Omron Sysmac Studio project TlsClientLib (Sysmac Studio 1.62.0.9, LibraryProject)
(* Develop simple TLS client library. *)

# Controller LIB: NX102-9000 version 1.64
Task Subsystem (priority 18, period or condition 10000): Example_SendLog
Library RingBufferLib 0.0.2 (contents left out)

TYPE stfreakjp\net\TlsClientContext : STRUCT
    Busy : BOOL;
    Active : BOOL;
    Error : BOOL;
    ErrorID : WORD;
    ErrorIDEx : DWORD;
    Port : UINT;
    Destination : STRING[256];
    DestinationPort : UINT;
    TLSSessionName : STRING[16];
    UseRecv : BOOL;
    UseSend : BOOL;
    UseWatcher : BOOL;
    UseTcpSocketOption : BOOL;
    OptionNodelay : BOOL;
    ConnectRetryTimes : UINT;
    ConnectRetryInterval : UINT;
    ConnectTimeout : UINT;
    WatchInterval : UINT;
    CtrlActive : BOOL;
    CtrlAllowSend : BOOL;
    CtrlAllowRecv : BOOL;
    Socket : _sSOCKET;
    TLSHandle : DWORD;
    Reconnecting : BOOL;
    Connected : BOOL;
    SendTimes : ULINT;
    SendSize : ULINT;
    RecvTimes : ULINT;
    RecvSize : ULINT;
END_STRUCT END_TYPE

PROGRAM README
RETURN;
(*

# About This Project
This project is for the development of the stream-oriented TLS clients: TlsClient, TlsSendClient, and TlsRecvClient.
TlsClient reads and writes TLS send/receive data to and from a ring buffer passed as a parameter.

The ring buffer utilizes RingBufferLib.
RingBufferLib is an implementation of a ring buffer for BYTE type arrays.
The RingBufferLib implementation can be used in multi-tasking environments without needing locks,
but only when there is a single reader and a single writer to the buffer.
TlsClient inherits this characteristic.

# About the Programs
This project includes the following examples.

* POU/Program/Example_SendLog
  This program uses TlsClient to send the contents of a logger's buffer to a remote location.
  Additionally, a debug-purpose TlsClient runs,
  monitoring and remotely sending the transmit buffer of the TlsClient that sends the logs.

Please refer to each program for usage steps.


# このプロジェクトについて
このプロジェクトは、ストリーム型TLSクライアントであるTlsClient/TlsSendClient/TlsRecvClientの開発用プロジェクトです。
TlsClientは、パラメータとして渡したリングバッファに対してTLSによる送受信データを読み書きします。
リングバッファは、RingBufferLibを使用します。
RingBufferLibはBYTE型配列を対象とするリングバッファの実装です。
RingBufferLibの実装は、バッファへの読み書きの主体がそれぞれ1つである時に限り、ロックを使用しなくてもマルチタスクに使用することができます。
TlsClientはその特性を引き継ぎます。

# プログラムについて
このプロジェクトは、以下の使用例を含みます。

* POU/プログラム/Example_SendLog
  TlsClientを使用してロガーのバッファ内容をリモートに送信します。
  また、ログを送信するTlsClientの送信バッファを監視してリモートに送信するデバッグ用のTlsClientが動作します。

使用手順については、各プログラムを確認してください。


For the parts to which I have rights, I follow POU/Program/LICENSE.
You are free to use and modify it, but we are not responsible for any damage or loss related to it.

(c) 2025 KITA Munemitsu

*)
END_PROGRAM

PROGRAM Example_SendLog
VAR CONSTANT
    LOG_SENDER_RESET_PAYLOAD : STRING[8] := '$$R$$L$$R$$L';
END_VAR
VAR
    REMOTE_ADDR : STRING[256];
    REMOTE_PORT : UINT;
    SPY_REMOTE_PORT : UINT;
    DEBUG_WRITE_REMOTE_PORT : UINT;
    DEBUG_READ_REMOTE_PORT : UINT;
    LOGGING_INTERVAL : UINT;
    iLogSenderTlsClient : stfreakjp\net\TlsClient;
    iLogSenderContext : stfreakjp\net\TlsClientContext;
    iLogSenderSendBufferContext : stfreakjp\buf\RingBufferContext;
    iLogSenderSendBuffer : ARRAY[0..8191] OF BYTE;
    iLogSenderRecvBufferContext : stfreakjp\buf\RingBufferContext;
    iLogSenderRecvBuffer : ARRAY[0..8191] OF BYTE;
    iLoggerWrittenTracker : stfreakjp\buf\RingBufferContext;
    iLoggerBufferContext : stfreakjp\buf\RingBufferContext;
    iLoggerBuffer : ARRAY[0..4095] OF BYTE;
    iPayload : ARRAY[0..4095] OF BYTE;
    iPayloadSize : UINT;
    iMsg : STRING[1024];
    iWaitTick : UINT;
    iSpySenderTlsClient : stfreakjp\net\TlsSendClient;
    iSpySenderClientContext : stfreakjp\net\TlsClientContext;
    iSpySendBufferContext : stfreakjp\buf\RingBufferContext;
    iSpySendBuffer : ARRAY[0..8191] OF BYTE;
    iSpyLogSenderSentTracker : stfreakjp\buf\RingBufferContext;
    iDebugReadSenderTlsClient : stfreakjp\net\TlsSendClient;
    iDebugReadSenderClientContext : stfreakjp\net\TlsClientContext;
    iDebugWriteSenderTlsClient : stfreakjp\net\TlsSendClient;
    iDebugWriteSenderClientContext : stfreakjp\net\TlsClientContext;
    iDebugWriteSenderBufferContext : stfreakjp\buf\RingBufferContext;
    iDebugWriteSenderBuffer : ARRAY[0..19999] OF BYTE;
    iDebugReadSenderBufferContext : stfreakjp\buf\RingBufferContext;
    iDebugReadSenderBuffer : ARRAY[0..19999] OF BYTE;
    iDebugLogSenderSendTracker : stfreakjp\buf\RingBufferContext;
    iToggleLogSend : BOOL;
END_VAR
(*

# About This Program
This program uses TlsClient to send the contents of a logger's buffer to a remote location.
Additionally, a debug-purpose TlsClient runs,
monitoring and remotely sending the transmit buffer of the TlsClient that sends the logs.

It is composed of the following:

* A logger that continuously writes logs.
* A log sender that sends logs written by the logger via TLS.
* A spy sender that monitors the log sender's transmission buffer and sends potentially transmitted logs via TLS.
* A debug sender that monitors read/write operations of the log sender's transmission buffer and sends each change via TLS.

# Usage Steps
Follow these steps to use the program.

1.  Adjust the project configuration to match your operating environment.   
    Match the controller model and ensure access to the network you intend to use.
  
2.  Adjust `POU/Program/Example_SendLog` to match your operating environment.   
    Change the value of the `REMOTE_ADDR` variable to the address of the device waiting for data.

3.  Start TLS endpoints on an appropriate device and wait for connections.
    You can find a reference PowerShell script in `POU/Program/SimpleTlsMonitor_ps1`.
	`StartMultiMonitors_ps1` is a PowerShell script that uses Windows Terminal to launch four TLS endpoints.

4.  Register TLS sessions on the controller.
    Register four TLS sessions with IDs 0-3.

5.  Run the program on the controller.   
    Transfer the program to the controller and start its execution.

6.  Confirm that data is sent to the listening TLS endpoints.


# このプログラムについて
このプログラムは、TlsClientを使用してロガーのバッファ内容をリモートに送信します。
また、ログを送信するTlsClientの送信バッファを監視してリモートに送信するデバッグ用のTlsClientが動作します。

以下によって構成します。

* ログを書き込み続けるロガー
* ロガーが書き込んだログをTLSで送信するログ送信クライアント
* ログ送信クライアントの送信バッファを監視して送信した可能性のあるログをTLSで送信するスパイ送信クライアント
* ログ送信クライアントの送信バッファの読み書きを監視して、それぞれの変化をTLSで送信するデバッグ送信クライアント

# 使用手順
このプログラムは、以下の手順で使用します。

1.  プロジェクトの構成を使用環境に合わせる
    コントローラの型式を合わせ、使用するネットワークにアクセスできるようにします。
  
2.  `POU/プログラム/Example_SendLog`を使用環境に合わせる
    `REMOTE_ADDR`変数の値をデータを待ち受ける端末のアドレスに変更します。
  
3.  適当な端末にTLSエンドポイントを立ち上げ待ち受ける
    `POU/プログラム/SimpleTlsMonitor_ps1`に参考のPowerShellスクリプトがあります。
	`StartMultiMonitors_ps1`は、Windows Terminalを使用して4つのTLSエンドポイントを立ち上げるPowerShellスクリプトです。

4.  コントローラにTLSセッションを登録する
    4つのTLSセッションをID 0-3で登録します。

5.  コントローラでプログラムを動作させる
    プログラムをコントローラに転送して動作させます。
  
6.  待ち受けているTLSエンドポイントにデータが送られてくることを確認する


(c) 2025 KITA Munemitsu

*)

// Change according to your environment.
IF P_First_Run THEN
	REMOTE_ADDR := 'YOUR_REMOTE_DEVICE';
	REMOTE_PORT := 12101;
	SPY_REMOTE_PORT := 12102;
	DEBUG_WRITE_REMOTE_PORT := 13101;
	DEBUG_READ_REMOTE_PORT := 13102;
	LOGGING_INTERVAL := 1;
END_IF;

IF P_First_Run THEN	
	// Setup Logger.
	Logger_init(Context:=iLoggerBufferContext,
				Buffer:=iLoggerBuffer);	

	// Setup Log sender.
	//
	// The log sender monitors the logger buffer and sends the written logs.
	//
	RingBuffer_init(Context:=iLogSenderSendBufferContext,
					Buffer:=iLogSenderSendBuffer);
	RingBuffer_init(Context:=iLogSenderRecvBufferContext,
					Buffer:=iLogSenderRecvBuffer);
	TlsClient_configure(Context:=iLogSenderContext,
						Activate:=TRUE,
						Destination:=REMOTE_ADDR,
						DestinationPort:=REMOTE_PORT,
						Port:=0,
						TLSSessionName:='TLSSession0',
						UseSend:=TRUE,
						UseRecv:=FALSE,
						UseWatcher:=TRUE,
						WatchInterval:=600,
						ConnectRetryTimes:=100,
						ConnectRetryInterval:=600);
	iLogSenderTlsClient.Enable := TRUE;
	// Tracks logger writes.
	RingBuffer_createWriteTracker(Target:=iLoggerBufferContext,
								  Tracker=>iLoggerWrittenTracker);

	// Setup Spy sender.
	//
    // The spy monitors the sender's transmit buffer and transmits any data that may have been sent.
	//
	RingBuffer_init(Context:=iSpySendBufferContext,
					Buffer:=iSpySendBuffer);
	TlsClient_configure(Context:=iSpySenderClientContext,
						Activate:=TRUE,
						Destination:=REMOTE_ADDR,
						DestinationPort:=SPY_REMOTE_PORT,
						Port:=0,
						TLSSessionName:='TLSSession1',
						UseSend:=TRUE,
						UseWatcher:=TRUE,
						WatchInterval:=600,
						ConnectRetryTimes:=100,
						ConnectRetryInterval:=600);
	iSpySenderTlsClient.Enable := TRUE;
	// Tracks reads of the log sender's send buffer.
	RingBuffer_createReadTracker(Target:=iLogSenderSendBufferContext,
								 Tracker=>iSpyLogSenderSentTracker);
 
    // Setup Debug senders.
	//
	// The debug sender monitors the input and output of the log sender's send buffer and sends the changes.
	//
	RingBuffer_init(Context:=iDebugWriteSenderBufferContext,
					Buffer:=iDebugWriteSenderBuffer);
	TlsClient_configure(Context:=iDebugWriteSenderClientContext,
						Activate:=TRUE,
						Destination:=REMOTE_ADDR,
						DestinationPort:=DEBUG_WRITE_REMOTE_PORT,
						Port:=0,
						TLSSessionName:='TLSSession2',
						UseSend:=TRUE,
						WatchInterval:=600,
						ConnectRetryTimes:=100,
						ConnectRetryInterval:=600);
	iDebugWriteSenderTlsClient.Enable := TRUE;
	
	RingBuffer_init(Context:=iDebugReadSenderBufferContext,
					Buffer:=iDebugReadSenderBuffer);
	TlsClient_configure(Context:=iDebugReadSenderClientContext,
						Activate:=TRUE,
						Destination:=REMOTE_ADDR,
						DestinationPort:=DEBUG_READ_REMOTE_PORT,
						Port:=0,
						TLSSessionName:='TLSSession3',
						UseSend:=TRUE,
						WatchInterval:=600,
						ConnectRetryTimes:=100,
						ConnectRetryInterval:=600);
	iDebugReadSenderTlsClient.Enable := TRUE;
	// Tracks the log sender's send buffer in and out.
	RingBuffer_createTracker(Target:=iLogSenderSendBufferContext,
							 Tracker=>iDebugLogSenderSendTracker);

	// Sends the log sender reset payload first.
	RingBuffer_writeString(Context:=iLogSenderSendBufferContext,
						   Buffer:=iLogSenderSendBuffer,
						   Value:=LOG_SENDER_RESET_PAYLOAD);

	iWaitTick := LOGGING_INTERVAL;
END_IF;

// Logging at regular intervals.
Dec(iWaitTick);
IF iWaitTick < 1 THEN
	iMsg := CONCAT('{"counter":', ULINT_TO_STRING(Get1usCnt()),
				   ',"timestamp":"', DtToString(GetTime()),
				   '"}$L');
	Logger_write(Context:=iLoggerBufferContext,
				 Buffer:=iLoggerBuffer,
				 Message:=iMsg);
	
	iWaitTick := LOGGING_INTERVAL;
END_IF;

IF iToggleLogSend THEN
	IF TlsClient_isAllowSend(Context:=iLogSenderContext) THEN
		TlsClient_disallowSend(Context:=iLogSenderContext);
	ELSE
		TlsClient_allowSend(Context:=iLogSenderContext);
	END_IF;
	iToggleLogSend := FALSE;
END_IF;

// Gets the difference of the logger buffer into the log sender's send buffer.
RingBuffer_pullWrite(Context:=iLogSenderSendBufferContext,
					 Buffer:=iLogSenderSendBuffer,
					 Tracker:=iLoggerWrittenTracker,
					 Tracked:=iLoggerBufferContext,
					 TrackedBuffer:=iLoggerBuffer);
iLogSenderTlsClient(Context:=iLogSenderContext,
					SendBufferContext:=iLogSenderSendBufferContext,
					SendBuffer:=iLogSenderSendBuffer,
					RecvBufferContext:=iLogSenderRecvBufferContext,
					RecvBuffer:=iLogSenderRecvBuffer);

// Gets the difference between the read data in the log sender's send buffer.
RingBuffer_pullRead(Context:=iSpySendBufferContext,
					Buffer:=iSpySendBuffer,
					Tracker:=iSpyLogSenderSentTracker,
					Tracked:=iLogSenderSendBufferContext,
					TrackedBuffer:=iLogSenderSendBuffer);
iSpySenderTlsClient(Context:=iSpySenderClientContext,
					SendBufferContext:=iSpySendBufferContext,
					SendBuffer:=iSpySendBuffer);

// Gets the read and write deferences of the log sender's send buffer.
RingBuffer_pull(WriteContext:=iDebugWriteSenderBufferContext,
				WriteBuffer:=iDebugWriteSenderBuffer,
				ReadContext:=iDebugReadSenderBufferContext,
				ReadBuffer:=iDebugReadSenderBuffer,
				Tracker:=iDebugLogSenderSendTracker,
				Tracked:=iLogSenderSendBufferContext,
				TrackedBuffer:=iLogSenderSendBuffer);
iDebugWriteSenderTlsClient(Context:=iDebugWriteSenderClientContext,
						   SendBufferContext:=iDebugWriteSenderBufferContext,
						   SendBuffer:=iDebugWriteSenderBuffer);
iDebugReadSenderTlsClient(Context:=iDebugReadSenderClientContext,
						  SendBufferContext:=iDebugReadSenderBufferContext,
						  SendBuffer:=iDebugReadSenderBuffer);
END_PROGRAM

PROGRAM SimpleTlsMonitor_ps1
RETURN;
(*

Below is a PowerShell script that starts a TLS server and waits for clients.


以下は、TLSサーバを立ち上げてクライアントを待ち受けるPowerShellスクリプトです。

```powershell:simple-tls-monitor.ps1
param(
    [Parameter(Mandatory=$false, Position=0)][int]$Port = 12101,
    [Parameter(Mandatory=$false, Position=1)][int]$ReadInterval = 50,
    [Parameter(Mandatory=$false, Position=2)][string]$Mode = 'jsonl',
    [Parameter(Mandatory=$false, Position=3)][string]$CertFriendlyName = 'TlsClientLibTest'
)

# Modify the following script and run it in PowerShell with administrator privileges
# to create a self-signed certificate.
#
# $param = @{
#    Type = 'SSLServerAuthentication'
#    DnsName = 'SET_YOUR_DOMAIN'
#    CertStoreLocation = 'Cert:\CurrentUser\My'
#    FriendlyName = 'TlsClientLibTest'
# }
# New-SelfSignedCertificate @params
#

$serverCert = Get-ChildItem -Path Cert:\CurrentUser\My
        | Where-Object { $_.FriendlyName -eq $CertFriendlyName }
if ($null -eq $serverCert) {
    Write-Host "No certs."
}

function Mode-Jsonl {
    param(
        [int]$Port,
        [int]$ReadInterval,
        [Object]$cert
    )
    $listenerEndPoint = New-Object IPEndpoint([System.Net.IPAddress]::Any, $Port)
    $tcpListener = New-Object System.Net.Sockets.TCPListener($listenerEndpoint)
    $client = $null
    $clientStream = $null
    $sslStream = $null
    $reader = $null
    $task = $null
    $entity = $null
    $prevEntity = $null

    try {
        $tcpListener.Start()
        while ($true) {
            # Wait for client connection.
            if ($null -eq $client) {
                if ($null -eq $task) {
                    $task = $tcpListener.AccepttcpClientAsync()
                }
                if (-not $task.Wait(200)) {
                    continue
                }
                $client = $task.GetAwaiter().GetResult()
                $clientStream = $client.GetStream()
                $sslStream = New-Object System.Net.Security.SslStream($clientStream, $false)
                $sslStream.AuthenticateAsServerAsync($cert, $false, [System.Security.Authentication.SslProtocols]::Tls12, $false).Wait()

                $reader = New-Object System.IO.StreamReader($sslStream)
                $task = $null
            }
            if ($reader.EndOfStream) {
                $reader.Close()
                $sslStream.Close()
                $clientStream.Close()
                $client.Close()
                $task = $null
                $reader = $null
                $clientStream = $null
                $client = $null
                $entity = $null
                $prevEntity = $null
                continue
            }

            # Waiting to receive data.
            try {
                if ($null -eq $task) {
                    $task = $reader.ReadLineAsync()
                }

                if (-not $task.Wait($ReadInterval)) {
                    continue
                }
                $entity = $task.GetAwaiter().GetResult();
                $task = $null
            }
            catch {
                Write-Host "error: $($_.Exception.Message)"
                $reader.Close()
                $clientStream.Close()
                $client.Close()
                $reader = $null
                $ClientStream = $null
                $client = $null
            }

            if ($null -ne $entity) {
                if ("" -eq $entity) {
                    if ("" -eq $prevEntity) {
                        Write-Host 'reset'
                    }
                } else {
                    try {
                        $entity | ConvertFrom-Json | Write-Host
                    }
                    catch {
                        Write-Host "error payload: ${entity}"
                    }
                }
            }

            $prevEntity = $entity
            $entity = $null
        }
    }
    catch {
        Write-Host "error: $($_.Exception.Message)"
    }
    finally {
        if ($client) {
            $reader.Close()
            $sslStream.Close()
            $clientStream.Close()
            $client.Close()
        }
        $tcpListener.Stop()
    }
}

function Mode-Raw {
    param(
        [string]$Port,
        [int]$ReadInterval,
        [Object]$cert
    )
    $listenerEndPoint = New-Object IPEndpoint([System.Net.IPAddress]::Any, $Port)
    $tcpListener = New-Object System.Net.Sockets.TCPListener($listenerEndpoint)
    $client = $null
    $clientStream = $null
    $reader = $null
    $task = $null
    $prevEntity = $null

    try {
        $tcpListener.Start()
        while ($true) {
            # Wait for client connection.
            if ($null -eq $client) {
                if ($null -eq $task) {
                    $task = $tcpListener.AcceptTcpClientAsync()
                }
                if (-not $task.Wait(200)) {
                    continue
                }

                $client = $task.GetAwaiter().GetResult();
                $clientStream = $client.GetStream()
                $sslStream = New-Object System.Net.Security.SslStream($clientStream, $false)
                $sslStream.AuthenticateAsServer($cert, $false, [System.Security.Authentication.SslProtocols]::Tls12, $false)
                $reader = New-Object System.IO.StreamReader($sslStream)
                $task = $null
            }
            if ($reader.EndOfStream) {
                $reader.Close()
                $sslStream.Close()
                $clientStream.Close()
                $client.Close()
                $task = $null
                $reader = $null
                $clientStream = $null
                $client = $null
                $entity = $null
                $prevEntity = $null
                continue
            }

            # Waiting to receive data.
            try {
                if ($null -eq $task) {
                    $task = $reader.ReadLineAsync()
                }

                if (-not $task.Wait($ReadInterval)) {
                    continue
                }
                $entity = $task.GetAwaiter().GetResult();
                $task = $null
            }
            catch {
                Write-Host "error: $($_.Exception.Message)"
                $reader.Close()
                $sslStream.Close()
                $clientStream.Close()
                $client.Close()
                $reader = $null
                $sslStream = $null
                $ClientStream = $null
                $client = $null
            }

            if ($null -ne $entity) {
                if ("" -eq $entity) {
                    if ("" -eq $prevEntity) {
                        Write-Host 'reset'
                    }
                } else {
                    $entity | Write-Host
                }
            }

            $prevEntity = $entity
            $entity = $null
        }
    }
    catch {
        Write-Host "error: $($_.Exception.Message)"
    }
    finally {
        if ($client) {
            $reader.Close()
            $sslStream.Close()
            $clientStream.Close()
            $client.Close()
        }
        $tcpListener.Stop()
    }
}

switch ( $Mode )
{
    Jsonl { Mode-Jsonl -Port $Port -ReadInterval $ReadInterval -cert $serverCert }
    Raw   { Mode-Raw -Port $Port -ReadInterval $ReadInterval -cert $serverCert }
}
```
*)
END_PROGRAM

PROGRAM StartMultiMonitors_ps1
RETURN;
(*

Below is a PowerShell script that launches four "simple-tls-monitor.ps" files in Windows Terminal.
Run this script while "simple-tls-monitor.ps1" is in the same folder.


以下は、Windows Terminalで4つの"simple-tls-monitor.ps"を立ち上げるPowerShellスクリプトです。
"simple-tls-monitor.ps1"が同じフォルダにある状態で実行します。

```powershell:start-multi-monitors.ps1
param(
    [Parameter(Mandatory=$false, Position=0)][int[]]$Ports = @(12101, 12102, 13101, 13102),
    [Parameter(Mandatory=$false, Position=1)][string]$Mode = 'jsonl',
    [Parameter(Mandatory=$false, Position=3)][string]$CertFriendlyName = 'TlsClientLibTest'
)

$scriptFile = "simple-tls-monitor.ps1"
$scriptDir = Split-Path -Parent $MyInvocation.MyCommand.Definition
$scriptPath = Join-Path $scriptDir $scriptFile
if (-not (Test-Path $scriptPath)) {
    Write-Error "error: Not fount '${scriptFile}' in '${scriptPath}'"
    exit 1
}

$wtCommandString = "pwsh.exe -NoExit -Command ""&{ & `"${scriptPath}`" -Port $($Ports[0]) -Mode `"${Mode}`" -CertFriendlyName `"${CertFriendlyName}`" }"" ; " + `
                   "split-pane -H pwsh.exe -NoExit -Command ""&{ & `"${scriptPath}`" -Port $($Ports[1]) -Mode `"${Mode}`" -CertFriendlyName `"${CertFriendlyName}`" }"" ; " + `
                   "split-pane -V pwsh.exe -NoExit -Command ""&{ & `"${scriptPath}`" -Port $($Ports[2]) -Mode `"${Mode}`" -CertFriendlyName `"${CertFriendlyName}`" }"" ; " + `
                   "split-pane -H pwsh.exe -NoExit -Command ""&{ & `"${scriptPath}`" -Port $($Ports[3]) -Mode `"${Mode}`" -CertFriendlyName `"${CertFriendlyName}`" }"""

# For debug.
# Write-Host "command: wt.exe $wtCommandString"

Start-Process -FilePath "wt.exe" -ArgumentList $wtCommandString
```
*)
END_PROGRAM

PROGRAM LICENSE
RETURN;
(*
The MIT License (MIT)

Copyright(c) 2025 KITA Munemitsu

Permission is hereby granted, free of charge, to any person obtaining a copy of this software and associated
documentation files (the “Software”), to deal in the Software without restriction, including without limitation
the rights to use, copy, modify, merge, publish, distribute, sublicense, and/or sell copies of the Software,
and to permit persons to whom the Software is furnished to do so, subject to the following conditions:

The above copyright notice and this permission notice shall be included in all copies or substantial portions of the Software.

THE SOFTWARE IS PROVIDED “AS IS”, WITHOUT WARRANTY OF ANY KIND, EXPRESS OR IMPLIED, INCLUDING BUT NOT
LIMITED TO THE WARRANTIES OF MERCHANTABILITY, FITNESS FOR A PARTICULAR PURPOSE AND NONINFRINGEMENT.
IN NO EVENT SHALL THE AUTHORS OR COPYRIGHT HOLDERS BE LIABLE FOR ANY CLAIM, DAMAGES OR OTHER LIABILITY,
WHETHER IN AN ACTION OF CONTRACT, TORT OR OTHERWISE, ARISING FROM, OUT OF OR IN CONNECTION WITH THE SOFTWARE
OR THE USE OR OTHER DEALINGS IN THE SOFTWARE.
*)
END_PROGRAM

FUNCTION stfreakjp\net\TlsClient_configure : BOOL
(* Initializes the TlsClientContext. *)
VAR_IN_OUT
    Context : stfreakjp\net\TlsClientContext;
END_VAR
VAR_INPUT
    Activate : BOOL := True;  (* Whether to activate the TLS client. Default is TRUE. *)
    Destination : STRING[256] := '';  (* Destination address. *)
    DestinationPort : UINT := 12101;  (* Destination port number. Default is 12101. *)
    Port : UINT := 0;  (* Port number of the TLS client socket. Default is 0 (Auto). *)
    TLSSessionName : STRING[16] := 'TLSSession0';  (* TLSSession name. Default is "TLSSession0". *)
    UseSend : BOOL := False;  (* Whether to use the Send feature. Default is FALSE. *)
    UseRecv : BOOL := False;  (* Whether to use the receive feature. Default is FALSE. *)
    UseWatcher : BOOL := False;  (* Whether to periodically check the connection status. Default is FALSE. *)
    WatchInterval : UINT := 300;  (* Interval between connection status checks. In 100ms increments. Defalt is 300 (30 sec). *)
    ConnectRetryTimes : UINT := 100;  (* Number of times the reconnect process will be attempted. Default is 100. *)
    ConnectRetryInterval : UINT := 300;  (* Interval between reconnection attempts. In 100ms increments. Defalt is 100 (10 sec). *)
    ConnectTimeout : UINT := 50;  (* Timeout waiting for connection. In 100ms increments. Default is 50 (5 sec). *)
    OptionNodelay : BOOL := False;  (* TCP_NODELAY option value. Default is FALSE. *)
END_VAR
(*

Initializes the TlsClientContext.


TlsClientContextを初期化する。


(c) 2025 KITA Munemitsu

*)

IF NOT EN THEN
	TlsClient_configure := FALSE;
	
	RETURN;
END_IF;

Context.CtrlActive := Activate;
Context.CtrlAllowSend := UseSend;
Context.CtrlAllowRecv := UseRecv;
Context.Destination := Destination;
Context.DestinationPort := DestinationPort;
Context.Port := Port;
Context.TLSSessionName := TLSSessionName;
Context.UseSend := UseSend;
Context.UseRecv := UseRecv;
Context.UseWatcher := UseWatcher;
Context.ConnectRetryTimes := ConnectRetryTimes;
Context.ConnectRetryInterval := ConnectRetryInterval;
Context.ConnectTimeout := ConnectTimeout;
Context.WatchInterval := WatchInterval;
Context.UseTcpSocketOption := OptionNodelay;
Context.OptionNodelay := OptionNodelay;

TlsClient_configure := TRUE;
END_FUNCTION

FUNCTION stfreakjp\net\TlsClient_activate : BOOL
(* Activates the TLS client. *)
VAR_IN_OUT
    Context : stfreakjp\net\TlsClientContext;  (* Target TlsClientContext. *)
END_VAR
(*

Activates the TLS client.


TLSクライアントを有効化する。


(c) 2025 KITA Munemitsu

*)

IF NOT EN THEN
	TlsClient_activate := FALSE;
	
	RETURN;
END_IF;
TlsClient_activate := TRUE;

Context.CtrlActive := TRUE;
END_FUNCTION

FUNCTION stfreakjp\net\TlsClient_deactivate : BOOL
(* Deactivates the TLS client. *)
VAR_IN_OUT
    Context : stfreakjp\net\TlsClientContext;  (* Target TlsClientContext. *)
END_VAR
(*

Deactivates the TLS client.


TLSクライアントを無効化する。


(c) 2025 KITA Munemitsu

*)

IF NOT EN THEN
	TlsClient_deactivate := FALSE;
	
	RETURN;
END_IF;
TlsClient_deactivate := TRUE;

Context.CtrlActive := FALSE;
END_FUNCTION

FUNCTION stfreakjp\net\TlsClient_isActive : BOOL  (* Whether the TCP client is active. *)
(* Returns whether the TLS client is active. *)
VAR_IN_OUT
    Context : stfreakjp\net\TlsClientContext;  (* Target TlsClientContext. *)
END_VAR
(*

Returns whether the TLS client is active.


TLSクライアントが有効かどうかを返す。


(c) 2025 KITA Munemitsu

*)

IF NOT EN THEN
	TlsClient_isActive := FALSE;
	
	RETURN;
END_IF;
TlsClient_isActive := Context.Active;
END_FUNCTION

FUNCTION stfreakjp\net\TlsClient_isAllowSend : BOOL
(* Returns whether send processing is allowed. *)
VAR_IN_OUT
    Context : stfreakjp\net\TlsClientContext;  (* Target TlsClientContext. *)
END_VAR
(*

Returns whether send processing is allowed.


送信処理を許可しているかどうかを返す。


(c) 2025 KITA Munemitsu

*)

IF NOT EN THEN
	TlsClient_isAllowSend := FALSE;
	
	RETURN;
END_IF;
TlsClient_isAllowSend := Context.CtrlAllowSend;
END_FUNCTION

FUNCTION stfreakjp\net\TlsClient_disallowSend : BOOL
(* Disallows execution of send processing. *)
VAR_IN_OUT
    Context : stfreakjp\net\TlsClientContext;  (* Target TlsClientContext. *)
END_VAR
(*

Disallows execution of send processing.


送信処理の実行を不許可にする。


(c) 2025 KITA Munemitsu

*)

IF NOT EN THEN
	TlsClient_disallowSend := FALSE;
	
	RETURN;
END_IF;
TlsClient_disallowSend := TRUE;

Context.CtrlAllowSend := FALSE;
END_FUNCTION

FUNCTION stfreakjp\net\TlsClient_allowSend : BOOL
(* Allows execution of send process. *)
VAR_IN_OUT
    Context : stfreakjp\net\TlsClientContext;  (* Target TlsClientContext. *)
END_VAR
(*

Allows execution of send process.


送信処理の実行を許可する。


(c) 2025 KITA Munemitsu

*)

IF NOT EN THEN
	TlsClient_allowSend := FALSE;
	
	RETURN;
END_IF;
TlsClient_allowSend := TRUE;

Context.CtrlAllowSend := TRUE;
END_FUNCTION

FUNCTION stfreakjp\net\TlsClient_isAllowRecv : BOOL
(* Returns whether to execute receive processing. *)
VAR_IN_OUT
    Context : stfreakjp\net\TlsClientContext;  (* Target TlsClientContext. *)
END_VAR
(*

Returns whether receive processing is allowed.


受信処理を許可しているかどうかを返す。


(c) 2025 KITA Munemitsu

*)

IF NOT EN THEN
	TlsClient_isAllowRecv := FALSE;
	
	RETURN;
END_IF;
TlsClient_isAllowRecv := Context.CtrlAllowRecv;
END_FUNCTION

FUNCTION stfreakjp\net\TlsClient_disallowRecv : BOOL
(* Disallows execution of receive processing. *)
VAR_IN_OUT
    Context : stfreakjp\net\TlsClientContext;  (* Target TlsClientContext. *)
END_VAR
(*

Disallows execution of receive processing.


受信処理の実行を不許可にする。


(c) 2025 KITA Munemitsu

*)

IF NOT EN THEN
	TlsClient_disallowRecv := FALSE;
	
	RETURN;
END_IF;
TlsClient_disallowRecv := TRUE;

Context.CtrlAllowRecv := FALSE;
END_FUNCTION

FUNCTION stfreakjp\net\TlsClient_allowRecv : BOOL
(* Allows execution of receive processing. *)
VAR_IN_OUT
    Context : stfreakjp\net\TlsClientContext;  (* Target TlsClientContext. *)
END_VAR
(*

Allows execution of receive processing.


受信処理の実行を許可する。


(c) 2025 KITA Munemitsu

*)

IF NOT EN THEN
	TlsClient_allowRecv := FALSE;
	
	RETURN;
END_IF;
TlsClient_allowRecv := TRUE;

Context.CtrlAllowRecv := TRUE;
END_FUNCTION

FUNCTION stfreakjp\net\TlsClient_isReconnecting : BOOL  (* Whether the TCP client is reconnecting. *)
(* Returns whether a TLS client is reconnecting. *)
VAR_IN_OUT
    Context : stfreakjp\net\TlsClientContext;  (* Target TlsClientContext. *)
END_VAR
(*

Returns whether a TLS client is reconnecting.


TLSクライアントが再接続中かどうかを返す。


(c) 2025 KITA Munemitsu

*)

IF NOT EN THEN
	TlsClient_isReconnecting := FALSE;
	
	RETURN;
END_IF;
TlsClient_isReconnecting := Context.Reconnecting;
END_FUNCTION

FUNCTION stfreakjp\net\TlsClient_getDestination : BOOL
(* Gets the current destination. *)
VAR_IN_OUT
    Context : stfreakjp\net\TlsClientContext;  (* Target TlsClientContext. *)
END_VAR
VAR_OUTPUT
    Destination : STRING[256];  (* Destination address. *)
    Port : UINT;  (* Destination port number. *)
END_VAR
(*

Gets the current destination.


現在の送信先を取得する。


(c) 2025 KITA Munemitsu

*)

IF NOT EN THEN
	Clear(Destination);
	Clear(Port);
	
	TlsClient_getDestination := FALSE;
	
	RETURN;
END_IF;

Destination := Context.Socket.DstAdr.IpAdr;
Port := Context.Socket.DstAdr.PortNo;

TlsClient_getDestination := TRUE;
END_FUNCTION

FUNCTION stfreakjp\net\TlsClient_getSource : BOOL
(* Gets the current source. *)
VAR_IN_OUT
    Context : stfreakjp\net\TlsClientContext;  (* Target TlsClientContext. *)
END_VAR
VAR_OUTPUT
    Source : STRING[256];  (* Address of the TLS client socket. *)
    Port : UINT;  (* Port number of the TLS client socket. *)
    TLSSessionName : STRING[16];  (* TLSSession name of the TLS client's connection. *)
END_VAR
(*

Gets the current source.


現在の送信元を取得する。


(c) 2025 KITA Munemitsu

*)

IF NOT EN THEN
	Clear(Source);
	Clear(Port);
	Clear(TLSSessionName);
	
	TlsClient_getSource := FALSE;
	
	RETURN;
END_IF;

Source := Context.Socket.SrcAdr.IpAdr;
Port := Context.Socket.SrcAdr.PortNo;
TLSSessionName := Context.TLSSessionName;

TlsClient_getSource := TRUE;
END_FUNCTION

FUNCTION stfreakjp\net\TlsClient_getError : BOOL  (* Whether the TCP client has an error. *)
(* Gets TLS client error information. *)
VAR_IN_OUT
    Context : stfreakjp\net\TlsClientContext;  (* Target TlsClientContext. *)
END_VAR
VAR_OUTPUT
    ErrorID : WORD;  (* Error ID. *)
    ErrorIDEx : DWORD;  (* Extended error ID. *)
END_VAR
(*

Gets TLS client error information.


TLSクライアントのエラー情報を取得する。


(c) 2025 KITA Munemitsu

*)

IF NOT EN
	OR NOT Context.Error
THEN
	Clear(ErrorID);
	Clear(ErrorIDEx);

	TlsClient_getError := FALSE;
	
	RETURN;
END_IF;

ErrorID := Context.ErrorID;
ErrorIDEx := Context.ErrorIDEx;

TlsClient_getError := TRUE;
END_FUNCTION

FUNCTION stfreakjp\net\TlsClient_hasError : BOOL  (* Whether the TCP client has an error. *)
(* Returns whether the TLS client has an error. *)
VAR_IN_OUT
    Context : stfreakjp\net\TlsClientContext;  (* Target TlsClientContext. *)
END_VAR
(*

Returns whether the TLS client has an error.


TLSクライアントでエラーが発生しているかどうかを返す。


(c) 2025 KITA Munemitsu

*)

IF NOT EN THEN
	TlsClient_hasError := FALSE;
	
	RETURN;
END_IF;

TlsClient_hasError := Context.Error;
END_FUNCTION

FUNCTION stfreakjp\net\TlsClient_getStat : BOOL  (* Whether the TCP client has an error. *)
(* Gets the status information of the TLS client. *)
VAR_IN_OUT
    Context : stfreakjp\net\TlsClientContext;  (* Target TlsClientContext. *)
END_VAR
VAR_OUTPUT
    SendTimes : ULINT;  (* Number of times sent since activation. *)
    SendSize : ULINT;  (* Bytes sent since activation. *)
    RecvTimes : ULINT;  (* Number of times received since activation. *)
    RecvSize : ULINT;  (* Bytes received since activation. *)
END_VAR
(*

Gets the status information of the TLS client.


TLSクライアントのステータス情報を取得する。


(c) 2025 KITA Munemitsu

*)

IF NOT EN
	OR NOT Context.Error
THEN
	Clear(SendTimes);
	Clear(SendSize);
	Clear(RecvTimes);
	Clear(RecvSize);

	TlsClient_getStat := FALSE;
	
	RETURN;
END_IF;

SendTimes := Context.SendTimes;
SendSize := Context.SendSize;
RecvTimes := Context.RecvTimes;
RecvSize := Context.RecvSize;

TlsClient_getStat := TRUE;
END_FUNCTION

FUNCTION Logger_write : BOOL
VAR
    iBinMsg : ARRAY[0..4095] OF BYTE;
    iBinMsgSize : UINT;
END_VAR
VAR_IN_OUT
    Context : stfreakjp\buf\RingBufferContext;
    Buffer : ARRAY[*] OF BYTE;
END_VAR
VAR_INPUT
    Message : STRING[1986] := '';
END_VAR
IF NOT EN THEN
	Logger_write := FALSE;
	
	RETURN;
END_IF;

iBinMsgSize
	:= StringToAry(In:=Message, AryOut:=iBinMsg[0]);
Logger_write
	:= \\stfreakjp\buf\RingBuffer_write(
						   Context:=Context,
						   Buffer:=Buffer,
						   In:=iBinMsg,
						   Head:=0,
						   Size:=iBinMsgSize,
						   AllowOverWrite:=TRUE);
END_FUNCTION

FUNCTION Logger_init : BOOL
VAR_IN_OUT
    Context : stfreakjp\buf\RingBufferContext;
    Buffer : ARRAY[*] OF BYTE;
END_VAR
IF NOT EN THEN
	Logger_init := FALSE;
	
	RETURN;
END_IF;

Logger_init
	:= \\stfreakjp\buf\RingBuffer_init(
						   Context:=Context,
						   Buffer:=Buffer);
END_FUNCTION

FUNCTION RingBuffer_writeString : BOOL
VAR
    iBinValue : ARRAY[0..4095] OF BYTE;
    iBinValueSize : UINT;
END_VAR
VAR_IN_OUT
    Context : stfreakjp\buf\RingBufferContext;
    Buffer : ARRAY[*] OF BYTE;
END_VAR
VAR_INPUT
    Value : STRING[1986] := '';
END_VAR
IF NOT EN THEN
	RingBuffer_writeString := FALSE;
	
	RETURN;
END_IF;

iBinValueSize
	:= StringToAry(In:=Value, AryOut:=iBinValue[0]);
RingBuffer_writeString
	:= \\stfreakjp\buf\RingBuffer_write(
						   Context:=Context,
						   Buffer:=Buffer,
						   In:=iBinValue,
						   Head:=0,
						   Size:=iBinValueSize,
						   AllowOverWrite:=TRUE);
END_FUNCTION

FUNCTION_BLOCK stfreakjp\net\TlsClient
(* TLS client that performs sending and receiving operations. *)
VAR
    iSktTCPConnect : SktTCPConnect;
    iSktClose : SktClose;
    iSktGetTCPStatus : SktGetTCPStatus;
    iSktSetOption : SktSetOption;
    iSktTLSConnect : SktTLSConnect;
    iSktTLSDisconnect : SktTLSDisconnect;
    iSktTLSWrite : SktTLSWrite;
    iSktTLSRead : SktTLSRead;
END_VAR
VAR CONSTANT
    STATE_INIT : UINT := 0;
    STATE_WAIT : UINT := 5;
    STATE_HALT : UINT := 9;
    STATE_ACTIVE : UINT := 10;
    STATE_RECONNECT : UINT := 20;
    STATE_CONNECT : UINT := 100;
    STATE_CLOSE : UINT := 110;
    STATE_CHANGE_DESTINATION : UINT := 120;
    STATE_FINALIZE : UINT := 900;
    STATE_DONE : UINT := 1000;
    STATE_SENDER_INIT : UINT := 0;
    STATE_SENDER_WAIT : UINT := 5;
    STATE_SENDER_ACTIVE : UINT := 10;
    STATE_SENDER_SEND : UINT := 200;
    STATE_SENDER_DONE : UINT := 1000;
    STATE_RECEIVER_INIT : UINT := 0;
    STATE_RECEIVER_WAIT : UINT := 5;
    STATE_RECEIVER_ACTIVE : UINT := 10;
    STATE_RECEIVER_RECV : UINT := 300;
    STATE_RECEIVER_DONE : UINT := 1000;
    STATE_WATCHER_INIT : UINT := 0;
    STATE_WATCHER_ACTIVE : UINT := 10;
    STATE_WATCHER_CHECK : UINT := 400;
    STATE_WATCHER_DONE : UINT := 1000;
END_VAR
VAR
    iState : UINT := 1001;
    iReturnState : UINT;
    iSocket : _sSOCKET;
    iTLSHandle : DWORD;
    iActive : BOOL;
    iError : BOOL;
    iErrorID : WORD;
    iErrorIDEx : DWORD;
    iConnectRetryTimes : UINT;
    iConnectRetryInterval : UINT;
    iConnectTimeout : UINT;
    iTimeoutTimer : _sTimer;
    iTimeout : BOOL;
    iWatchInterval : UINT;
    iWillTcpEstablished : BOOL;
    iTcpStatus : _eCONNECTION_STATE;
    iOptionNodelay : BOOL;
    iRetryTimes : UINT;
    iRetryInterval : UINT;
    iRetryTimer : _sTimer;
    iDoRetry : BOOL;
    iStateSender : UINT := 1000;
    iSendData : ARRAY[0..1999] OF BYTE;
    iSendDataSize : UINT;
    iSenderError : BOOL;
    iSenderErrorID : WORD;
    iSenderWaitTick : UINT;
    iStateReceiver : UINT := 1000;
    iRecvData : ARRAY[0..1999] OF BYTE;
    iRecvDataSize : UINT;
    iReceiverError : BOOL;
    iReceiverErrorID : WORD;
    iReceiverWaitTick : UINT;
    iStateWatcher : UINT := 1000;
    iWatcherError : BOOL;
    iWatcherErrorID : WORD;
    iWatchTimer : _sTimer;
    iWatchDoCheck : BOOL;
    iB : DWORD;
    iHere : BOOL;
END_VAR
VAR_INPUT
    Enable : BOOL;  (* Enable TlsClient FB. *)
END_VAR
VAR_IN_OUT
    Context : stfreakjp\net\TlsClientContext;  (* TlsClientContext to process. *)
    SendBufferContext : stfreakjp\buf\RingBufferContext;  (* RingBufferContext for the sent data. *)
    SendBuffer : ARRAY[*] OF BYTE;  (* Buffer for sent data. *)
    RecvBufferContext : stfreakjp\buf\RingBufferContext;  (* RingBufferContext for the received data. *)
    RecvBuffer : ARRAY[*] OF BYTE;  (* Buffer for received data. *)
END_VAR
VAR_OUTPUT
    Busy : BOOL;  (* Whether the TlsClient is running. *)
    Done : BOOL;  (* Whether the TlsClient has completed processing. *)
END_VAR
(*

TLS client that performs sending and receiving operations.


送受信処理を行うTLSクライアント。

(c) 2025 KITA Munemitsu

*)

Done := FALSE;
IF Enable AND NOT Busy THEN
	iState := STATE_INIT;
	
	Busy := TRUE;
END_IF;

CASE iState OF
	// STATE_INIT
	0:
		iSktTCPConnect.Execute := FALSE;
		iSktClose.Execute := FALSE;
		iSktGetTCPStatus.Execute := FALSE;
		iSktTLSConnect.Execute := FALSE;
		iSktTLSDisconnect.Execute := FALSE;
		iSktTLSRead.Execute := FALSE;
		iSktTLSWrite.Execute := FALSE;

		Clear(iActive);
		Clear(iSocket);
		Clear(iTLSHandle);
		Clear(iError);
		Clear(iErrorID);
		Clear(iErrorIDEx);
		
		Clear(Context.Active);
		Clear(Context.Busy);
		Clear(Context.Error);
		Clear(Context.ErrorID);
		Clear(Context.ErrorIDEx);
		Clear(Context.Connected);
		Clear(Context.Reconnecting);
		Clear(Context.Socket);
		Clear(Context.TLSHandle);
		Clear(Context.SendTimes);
		Clear(Context.SendSize);
		Clear(Context.RecvTimes);
		Clear(Context.RecvSize);

		iWillTcpEstablished := TRUE;
		iConnectRetryTimes := Context.ConnectRetryTimes;
		iConnectRetryInterval := MAX(UINT#100, Context.ConnectRetryInterval);
		iConnectTimeout := MAX(UINT#10, Context.ConnectTimeout);
		iWatchInterval := MAX(UINT#100, Context.WatchInterval);
		iOptionNodelay := Context.OptionNodelay;

		iState := STATE_WAIT;
		
	// STATE_WAIT
	5:
		IF Context.CtrlActive THEN
			iReturnState := iState + 1;
			iState := STATE_CONNECT;
		END_IF;
	6:
		IF iError THEN			
			Context.Error := TRUE;
			Context.ErrorID := iErrorID;
			Context.ErrorIDEx := iErrorIDEx;
			
			IF iConnectRetryTimes < 1 THEN
				iState := STATE_HALT;
			ELSE
				iReturnState := STATE_RECONNECT;
				iState := STATE_CLOSE;
			END_IF;
		ELSE
			iActive := TRUE;
			IF Context.UseSend THEN
				iStateSender := STATE_SENDER_INIT;
			END_IF;
			IF Context.UseRecv THEN
				iStateReceiver := STATE_RECEIVER_INIT;
			END_IF;
			IF Context.UseWatcher THEN
				iStateWatcher := STATE_WATCHER_INIT;
			END_IF;
			
			iState := STATE_ACTIVE;
		END_IF;
			
	// STATE_HALT
	9:
		IF NOT (Context.CtrlActive AND Enable) THEN
			iState := STATE_FINALIZE;
		END_IF;
	
	// STATE_ACTIVE
	10:
		IF NOT (Context.CtrlActive AND Enable) THEN
			iState := STATE_FINALIZE;
		ELSIF iSenderError THEN
			Context.Error := TRUE;
			Context.ErrorID := iSenderErrorID;
			Context.ErrorIDEx := SHL(WORD_TO_DWORD(iSenderErrorID), 16) OR UINT_TO_DWORD(STATE_SENDER_SEND);
			iActive := FALSE;
			
			IF iConnectRetryTimes < 1 THEN
				iReturnState := STATE_HALT;
				iState := STATE_CLOSE;
			ELSE
				iReturnState := STATE_RECONNECT;
				iState := STATE_CLOSE;
			END_IF;
		ELSIF iReceiverError THEN
			Context.Error := TRUE;
			Context.ErrorID := iReceiverErrorID;
			Context.ErrorIDEx := SHL(WORD_TO_DWORD(iReceiverErrorID), 16) OR UINT_TO_DWORD(STATE_RECEIVER_RECV);
			iActive := FALSE;
			
			IF iConnectRetryTimes < 1 THEN
				iReturnState := STATE_HALT;
				iState := STATE_CLOSE;
			ELSE
				iReturnState := STATE_RECONNECT;
				iState := STATE_CLOSE;
			END_IF;
		ELSIF iWatcherError THEN
			Context.Error := TRUE;
			Context.ErrorID := iWatcherErrorID;
			Context.ErrorIDEx := SHL(WORD_TO_DWORD(iWatcherErrorID), 16) OR UINT_TO_DWORD(STATE_WATCHER_CHECK);
			iActive := FALSE;
			
			IF iConnectRetryTimes < 1 THEN
				iReturnState := STATE_HALT;
				iState := STATE_CLOSE;
			ELSE
				iReturnState := STATE_RECONNECT;
				iState := STATE_CLOSE;
			END_IF;
		ELSIF NOT iWillTcpEstablished THEN
			iActive := FALSE;
			
			IF iConnectRetryTimes < 1 THEN
				iReturnState := STATE_HALT;
				iState := STATE_CLOSE;
			ELSE
				iReturnState := STATE_RECONNECT;
				iState := STATE_CLOSE;
			END_IF;
		END_IF;		

	// STATE_RECONNECT
	20:
		iRetryTimes := iConnectRetryTimes;
		Timer(In:=FALSE,
			  PT:=iConnectRetryInterval,
			  TimerDat:=iRetryTimer,
			  Q=>iDoRetry);
		Context.Reconnecting := TRUE;
		
		Inc(iState);
	21:
		Timer(In:=TRUE,
			  PT:=iConnectRetryInterval,
			  TimerDat:=iRetryTimer,
			  Q=>iDoRetry);
		IF NOT (Context.CtrlActive AND Enable) THEN
			Context.Reconnecting := FALSE;
			
			iState := STATE_FINALIZE;
		ELSIF iDoRetry THEN
			iReturnState := iState + 1;
			iState := STATE_CONNECT;
		END_IF;
	22:
		IF iError THEN
			Dec(iRetryTimes);
			IF iRetryTimes < 1 THEN				
				iState := iState + 7;
			ELSE
				Timer(In:=FALSE,
					  PT:=iConnectRetryInterval,
					  TimerDat:=iRetryTimer,
					  Q=>iDoRetry);
				
				Dec(iState);
			END_IF;
		ELSE
			iState := iState + 7;
		END_IF;
	29:
		IF iError THEN
			Context.Error := TRUE;
			Context.ErrorID := iErrorID;
			Context.ErrorIDEx := iErrorIDEx;
			
			iState := STATE_HALT;
		ELSE
			Clear(Context.Error);
			Clear(Context.ErrorID);
			Clear(Context.ErrorIDEx);
			
			iActive := TRUE;
			IF Context.UseSend THEN
				iStateSender := STATE_SENDER_INIT;
			END_IF;
			IF Context.UseRecv THEN
				iStateReceiver := STATE_RECEIVER_INIT;
			END_IF;
			IF Context.UseWatcher THEN
				iStateWatcher := STATE_WATCHER_INIT;
			END_IF;

			iState := STATE_ACTIVE;
		END_IF;
		Context.Reconnecting := FALSE;
		
	// STATE_CONNECT
	100:
		Clear(iError);
		Clear(iErrorID);
		Clear(iErrorIDEx);
		Timer(In:=FALSE,
			  PT:=iConnectTimeout,
			  TimerDat:=iTimeoutTimer);
		
		iSktTCPConnect.DstAdr := Context.Destination;
		iSktTCPConnect.DstTcpPort := Context.DestinationPort;
		iSktTCPConnect.SrcTcpPort := Context.Port;
		iSktTCPConnect.Execute := TRUE;

		Inc(iState);
	101:
		Timer(In:=TRUE,
			  PT:=iConnectTimeout,
			  TimerDat:=iTimeoutTimer,
			  Q=>iTimeout);
		IF iSktTCPConnect.Done OR iSktTCPConnect.Error THEN
			iSktTCPConnect.Execute := FALSE;
			
			IF iSktTCPConnect.Error THEN
				iError := TRUE;
				iErrorID := iSktTCPConnect.ErrorID;
				iErrorIDEx := SHL(WORD_TO_DWORD(iErrorID), 16) OR UINT_TO_DWORD(iState);
				
				iState := iState + 8;
			ELSE
				iSocket := iSktTCPConnect.Socket;
				Context.Socket := iSocket;

				Inc(iState);
			END_IF;
		ELSIF iTimeout THEN
			iSktTCPConnect.Execute := FALSE;
			
			iError := TRUE;
			iErrorID := WORD#16#2006; // Socket timeout.
			iErrorIDEx := SHL(WORD_TO_DWORD(iErrorID), 16) OR UINT_TO_DWORD(iState);
			
			iState := iState + 8;
		END_IF;
	102:
		IF NOT Context.UseTcpSocketOption THEN
			iState := iState + 3;
		ELSE
			Inc(iState);
		END_IF;
	103:
		iSktSetOption(Execute:=FALSE,
					  OptionType:=_eSKT_OPTION_TYPE#_TCP_NODELAY,
					  OptionParam:=iOptionNodelay);

		Inc(iState);
	104:
		iSktSetOption(Execute:=TRUE,
					  Socket:=iSocket,
					  OptionType:=_eSKT_OPTION_TYPE#_TCP_NODELAY,
					  OptionParam:=iOptionNodelay);

		IF iSktSetOption.Done OR iSktSetOption.Error THEN
			iSktSetOption.Execute := FALSE;

			IF iSktSetOption.Error THEN
				iError := TRUE;
				iErrorID := iSktSetOption.ErrorID;
				iErrorIDEx := SHL(WORD_TO_DWORD(iErrorID), 16) OR UINT_TO_DWORD(iState);
				
				iState := iState + 5;
			ELSE
				Inc(iState);
			END_IF;
		END_IF;
	105:
		iSktTLSConnect.Socket := iSocket;
		iSktTLSConnect.TLSSessionName := Context.TLSSessionName;
		iSktTLSConnect.Execute := TRUE;
		
		Inc(iState);
	106:
		IF iSktTLSConnect.Done OR iSktTLSConnect.Error THEN
			iSktTLSConnect.Execute := FALSE;
			
			IF iSktTLSConnect.Error THEN
				iError := TRUE;
				iErrorID := iSktTLSConnect.ErrorID;
				iErrorIDEx := SHL(WORD_TO_DWORD(iErrorID), 16) OR UINT_TO_DWORD(iState);	
			ELSE
				iTLSHandle := iSktTLSConnect.Handle;
				Context.TLSHandle := iTLSHandle;
			END_IF;
			
			iState := iState + 3;
		END_IF;
	109:
		Context.Connected := NOT iError;
		
		iState := iReturnState;

	// STATE_CLOSE
	110:
		Clear(iError);
		Clear(iErrorID);
		Clear(iErrorIDEx);
	
		iSktTLSDisconnect.Handle := iTLSHandle;
		iSktTLSDisconnect.Execute := TRUE;
		
		Inc(iState);
	111:
		IF iSktTLSDisconnect.Done OR iSktTLSDisconnect.Error THEN
			iSktTLSDisconnect.Execute := FALSE;
			
			IF iSktTLSDisconnect.Error THEN
				iError := TRUE;
				iErrorID := iSktTLSDisconnect.ErrorID;
				iErrorIDEx := SHL(WORD_TO_DWORD(iErrorID), 16) OR UINT_TO_DWORD(iState);
			END_IF;
			
			Inc(iState);
		END_IF;
	112:
		iSktClose.Socket := iSocket;
		iSktClose.Execute := TRUE;
		
		Inc(iState);
	113:
		IF iSktClose.Done OR iSktClose.Error THEN
			iSktClose.Execute := FALSE;
			
			IF iSktClose.Error AND NOT iError THEN
				iError := TRUE;
				iErrorID := iSktClose.ErrorID;
				iErrorIDEx := SHL(WORD_TO_DWORD(iErrorID), 16) OR UINT_TO_DWORD(iState);
			END_IF;
			
			iState := iState + 6;
		END_IF;
	119:
		Context.Connected := FALSE;
		
		iState := iReturnState;
		
	// STATE_FINALIZE
	900:
		iActive := FALSE;
		
		Inc(iState);
	901:
		IF iStateSender = STATE_SENDER_DONE THEN
			IF iSenderError AND NOT Context.Error THEN
				Context.Error := TRUE;
				Context.ErrorID := iSenderErrorID;
				Context.ErrorIDEx := SHL(WORD_TO_DWORD(iSenderErrorID), 16) OR UINT_TO_DWORD(iState);
			END_IF;
			
			Inc(iState);
		END_IF;
	902:
		IF iStateReceiver = STATE_RECEIVER_DONE THEN
			IF iReceiverError AND NOT Context.Error THEN
				Context.Error := TRUE;
				Context.ErrorID := iReceiverErrorID;
				Context.ErrorIDEx := SHL(WORD_TO_DWORD(iReceiverErrorID), 16) OR UINT_TO_DWORD(iState);
			END_IF;
			
			Inc(iState);
		END_IF;
	903:
		IF iStateWatcher = STATE_WATCHER_DONE THEN
			IF iWatcherError AND NOT Context.Error THEN
				Context.Error := TRUE;
				Context.ErrorID := iWatcherErrorID;
				Context.ErrorIDEx := SHL(WORD_TO_DWORD(iWatcherErrorID), 16) OR UINT_TO_DWORD(iState);
			END_IF;
			
			Inc(iState);
		END_IF;
	904:
		IF Context.Connected THEN
			iReturnState := iState + 1;
			iState := STATE_CLOSE;
		ELSE
			iState := iState + 5;
		END_IF;
	905:
		IF iError AND NOT Context.Error THEN
			Context.Error := TRUE;
			Context.ErrorID := iErrorID;
			Context.ErrorIDEx := iErrorIDEx;
		END_IF;
		
		iState := iState + 4;
	909:
		iState := STATE_DONE;
	
	// STATE_DONE
	1000:
		Done := TRUE;
		Busy := FALSE;
		
		Inc(iState);
END_CASE;

CASE iStateSender OF
	// STATE_SENDER_INIT
	0:
		iSktTLSWrite.Execute := FALSE;

		Clear(iSenderError);
		Clear(iSenderErrorID);
		
		iStateSender := STATE_SENDER_ACTIVE;
				
	// STATE_SENDER_ACTIVE
	10:
		IF NOT iActive THEN
			iStateSender := STATE_SENDER_DONE;
		ELSIF \\stfreakjp\buf\RingBuffer_isReadable(
								  Context:=SendBufferContext)
		THEN
			iStateSender := STATE_SENDER_SEND;
		END_IF;
	
	// STATE_SENDER_SEND
	200:
		IF Context.CtrlAllowSend THEN
			\\stfreakjp\buf\RingBuffer_peekFully(
								Context:=SendBufferContext,
								Buffer:=SendBuffer,
								Out:=iSendData,
								Head:=0,
								ReadSize=>iSendDataSize);
			
			IF iSendDataSize < 1 THEN
				iStateSender := STATE_SENDER_ACTIVE;
			ELSE
				iSktTLSWrite.Handle := iTLSHandle;
				iSktTLSWrite.SendDatSize := iSendDataSize;
				iSktTLSWrite.Execute := TRUE;
				
				Inc(iStateSender);
			END_IF;
		ELSIF NOT iActive THEN
			iStateSender := STATE_SENDER_DONE;
		END_IF;
	201:
		IF iSktTLSWrite.Done OR iSktTLSWrite.Error THEN
			iSktTLSWrite.Execute := FALSE;
			
			IF iSktTLSWrite.Error THEN
				iSenderErrorID := iSktTLSWrite.ErrorID;
				CASE WORD_TO_UINT(iSenderErrorID) OF
					// Socket communication resource over.
					16#2008:
						iSenderWaitTick
							:= MAX(UINT#10, TO_UINT(iSendDataSize MOD 50));
						
						Inc(iStateSender);
				ELSE
					iSenderError := TRUE;
					
					iStateSender := STATE_SENDER_DONE;
				END_CASE;
			ELSE
				\\stfreakjp\buf\RingBuffer_consume(
									Context:=SendBufferContext,
									Buffer:=SendBuffer,
									Size:=iSendDataSize);
				
				Context.SendSize := Context.SendSize + iSendDataSize;
				Inc(Context.SendTimes);
				
				Dec(iStateSender);
			END_IF;
		END_IF;
	202:
		Dec(iSenderWaitTick);
		IF NOT iActive THEN
			iSenderError := TRUE;

			iStateSender := STATE_SENDER_DONE;
		ELSIF NOT Context.CtrlAllowSend THEN
			iStateSender := iStateSender - 2;
		ELSIF iSenderWaitTick < 1 THEN
			iSktTLSWrite.Execute := TRUE;
			
			Dec(iStateSender);
		END_IF;
	
	// STATE_SENDER_DONE
	// 1000:
END_CASE;

CASE iStateReceiver OF
	// STATE_RECEIVER_INIT
	0:
		iSktTLSRead.Execute := FALSE;

		Clear(iReceiverError);
		Clear(iReceiverErrorID);
		
		iStateReceiver := STATE_RECEIVER_ACTIVE;
				
	// STATE_RECEIVER_ACTIVE
	10:
		IF NOT iActive THEN
			iStateReceiver := STATE_RECEIVER_DONE;
		ELSIF \\stfreakjp\buf\RingBuffer_isWritable(
								  Context:=RecvBufferContext)
		THEN
			iStateReceiver := STATE_RECEIVER_RECV;
		END_IF;
	
	// STATE_RECEIVER_RECV
	300:
		IF Context.CtrlAllowRecv THEN
			iSktTLSRead.TimeOut := 0;
			iSktTLSRead.Handle := iTLSHandle;
			iSktTLSRead.Execute := TRUE;
		
			Inc(iStateReceiver);
		ELSIF NOT iActive THEN
			iStateReceiver := STATE_RECEIVER_DONE;
		END_IF;
	301:
		IF NOT iActive THEN
			iSktTLSRead.Execute := FALSE;
			
			iStateReceiver := STATE_RECEIVER_DONE;
		ELSIF NOT Context.CtrlAllowRecv THEN
			iSktTLSRead.Execute := FALSE;
			
			Dec(iStateReceiver);
		ELSIF iSktTLSRead.Done OR iSktTLSRead.Error THEN
			iSktTLSRead.Execute := FALSE;
			
			IF iSktTLSRead.Error THEN
				iReceiverErrorID := iSktTLSRead.ErrorID;
				CASE WORD_TO_UINT(iReceiverErrorID) OF
					// Socket communication resource over.
					16#2008:
						iReceiverWaitTick := UINT#10;
						
						iStateReceiver := iStateReceiver + 2;
				ELSE
					iReceiverError := TRUE;
					
					iStateReceiver := STATE_RECEIVER_DONE;
				END_CASE;
			ELSE
				iRecvDataSize := iSktTLSRead.RcvSize;
				Context.RecvSize := Context.RecvSize + iRecvDataSize;
				Inc(Context.RecvTimes);
				
				IF \\stfreakjp\buf\RingBuffer_write(
									   Context:=RecvBufferContext,
									   Buffer:=RecvBuffer,
									   In:=iRecvData,
									   Head:=0,
									   Size:=iRecvDataSize)
				THEN					
					Dec(iStateReceiver);
				ELSE					
					Inc(iStateReceiver);
				END_IF;
			END_IF;
		END_IF;
	302:
		IF NOT iActive THEN
			iStateReceiver := STATE_RECEIVER_DONE;
		ELSIF \\stfreakjp\buf\RingBuffer_write(
								  Context:=RecvBufferContext,
								  Buffer:=RecvBuffer,
								  In:=iRecvData,
								  Head:=0,
								  Size:=iRecvDataSize)
		THEN
			iStateReceiver := iStateReceiver - 2;
		END_IF;
	303:
		Dec(iReceiverWaitTick);
		IF NOT iActive THEN
			iReceiverError := TRUE;

			iStateReceiver := STATE_RECEIVER_DONE;
		ELSIF iReceiverWaitTick < 1 THEN
			iStateReceiver := iStateReceiver - 3;
		END_IF;
	
	// STATE_RECEIVER_DONE
	// 1000:
END_CASE;

CASE iStateWatcher OF
	// STATE_WATCHER_INIT
	0:
		iSktGetTCPStatus.Execute := FALSE;
		
		Clear(iWatcherError);
		Clear(iWatcherErrorID);

		Timer(In:=FALSE,
			  PT:=iWatchInterval,
			  TimerDat:=iWatchTimer);
		
		iStateWatcher := STATE_WATCHER_ACTIVE;
		
	// STATE_WATCHER_ACTIVE
	10:
		Timer(In:=TRUE,
			  PT:=iWatchInterval,
			  TimerDat:=iWatchTimer,
			  Q=>iWatchDoCheck);
		IF NOT iActive THEN
			iStateWatcher := STATE_WATCHER_DONE;
		ELSIF iWatchDoCheck THEN
			iStateWatcher := STATE_WATCHER_CHECK;
		END_IF;
	
	// STATE_WATCHER_CHECK
	400:
		iSktGetTCPStatus.Socket := iSocket;
		iSktGetTCPStatus.Execute := TRUE;
		
		Inc(iStateWatcher);
	401:
		IF iSktGetTCPStatus.Done OR iSktGetTCPStatus.Error THEN
			iSktGetTCPStatus.Execute := FALSE;
			
			IF iSktGetTCPStatus.Error THEN
				iWatcherError := TRUE;
				iWatcherErrorID := iSktGetTCPStatus.ErrorID;
				
				iStateWatcher := STATE_WATCHER_DONE;
			ELSE
				iTcpStatus := iSktGetTCPStatus.TcpStatus;
				CASE iTcpStatus OF
					_eCONNECTION_STATE#_ESTABLISHED:
						iWillTcpEstablished := TRUE;
				ELSE
					iWillTcpEstablished := FALSE;
				END_CASE;
				
				Timer(In:=FALSE,
					  PT:=iWatchInterval,
					  TimerDat:=iWatchTimer);
				
				iStateWatcher := STATE_WATCHER_ACTIVE;
			END_IF;
		END_IF;
	
	// STATE_WATCHER_DONE
	// 1000:
END_CASE;

iSktTCPConnect();
iSktClose();
iSktGetTCPStatus();
iSktTLSConnect();
iSktTLSDisconnect();
iSktTLSWrite(SendDat:=iSendData[0]);
iSktTLSRead(RcvDat:=iRecvData[0]);

Context.Active := iActive;
Context.Busy := Busy;
END_FUNCTION_BLOCK

FUNCTION_BLOCK stfreakjp\net\TlsSendClient
(* TLS client that performs sending and receiving operations. *)
VAR
    iSktTCPConnect : SktTCPConnect;
    iSktTLSConnect : SktTLSConnect;
    iSktClose : SktClose;
    iSktTLSDisconnect : SktTLSDisconnect;
    iSktGetTCPStatus : SktGetTCPStatus;
    iSktSetOption : SktSetOption;
    iSktTLSWrite : SktTLSWrite;
END_VAR
VAR CONSTANT
    STATE_INIT : UINT := 0;
    STATE_WAIT : UINT := 5;
    STATE_HALT : UINT := 9;
    STATE_ACTIVE : UINT := 10;
    STATE_RECONNECT : UINT := 20;
    STATE_CONNECT : UINT := 100;
    STATE_CLOSE : UINT := 110;
    STATE_CHANGE_DESTINATION : UINT := 120;
    STATE_FINALIZE : UINT := 900;
    STATE_DONE : UINT := 1000;
    STATE_SENDER_INIT : UINT := 0;
    STATE_SENDER_WAIT : UINT := 5;
    STATE_SENDER_ACTIVE : UINT := 10;
    STATE_SENDER_SEND : UINT := 200;
    STATE_SENDER_DONE : UINT := 1000;
    STATE_WATCHER_INIT : UINT := 0;
    STATE_WATCHER_ACTIVE : UINT := 10;
    STATE_WATCHER_CHECK : UINT := 400;
    STATE_WATCHER_DONE : UINT := 1000;
END_VAR
VAR
    iState : UINT := 1001;
    iReturnState : UINT;
    iSocket : _sSOCKET;
    iTLSHandle : DWORD;
    iActive : BOOL;
    iError : BOOL;
    iErrorID : WORD;
    iErrorIDEx : DWORD;
    iConnectRetryTimes : UINT;
    iConnectRetryInterval : UINT;
    iConnectTimeout : UINT;
    iTimeoutTimer : _sTimer;
    iTimeout : BOOL;
    iWatchInterval : UINT;
    iWillTcpEstablished : BOOL;
    iTcpStatus : _eCONNECTION_STATE;
    iOptionNodelay : BOOL;
    iRetryTimes : UINT;
    iRetryInterval : UINT;
    iRetryTimer : _sTimer;
    iDoRetry : BOOL;
    iStateSender : UINT := 1000;
    iSendData : ARRAY[0..1999] OF BYTE;
    iSendDataSize : UINT;
    iSenderError : BOOL;
    iSenderErrorID : WORD;
    iSenderWaitTick : UINT;
    iStateWatcher : UINT := 1000;
    iWatcherError : BOOL;
    iWatcherErrorID : WORD;
    iWatchTimer : _sTimer;
    iWatchDoCheck : BOOL;
END_VAR
VAR_INPUT
    Enable : BOOL;  (* Enable TlsClient FB. *)
END_VAR
VAR_IN_OUT
    Context : stfreakjp\net\TlsClientContext;  (* TlsClientContext to process. *)
    SendBufferContext : stfreakjp\buf\RingBufferContext;  (* RingBufferContext for the sent data. *)
    SendBuffer : ARRAY[*] OF BYTE;  (* Buffer for sent data. *)
END_VAR
VAR_OUTPUT
    Busy : BOOL;  (* Whether the TlsClient is running. *)
    Done : BOOL;  (* Whether the TlsClient has completed processing. *)
END_VAR
(*

TLS client that performs sending operations.


送信処理を行うTLSクライアント。

(c) 2025 KITA Munemitsu

*)

Done := FALSE;
IF Enable AND NOT Busy THEN
	iState := STATE_INIT;
	
	Busy := TRUE;
END_IF;

CASE iState OF
	// STATE_INIT
	0:
		iSktTCPConnect.Execute := FALSE;
		iSktClose.Execute := FALSE;
		iSktGetTCPStatus.Execute := FALSE;
		iSktTLSConnect.Execute := FALSE;
		iSktTLSDisconnect.Execute := FALSE;
		iSktTLSWrite.Execute := FALSE;

		Clear(iActive);
		Clear(iSocket);
		Clear(iTLSHandle);
		Clear(iError);
		Clear(iErrorID);
		Clear(iErrorIDEx);
		
		Clear(Context.Active);
		Clear(Context.Busy);
		Clear(Context.Error);
		Clear(Context.ErrorID);
		Clear(Context.ErrorIDEx);
		Clear(Context.Connected);
		Clear(Context.Reconnecting);
		Clear(Context.Socket);
		Clear(Context.TLSHandle);
		Clear(Context.SendTimes);
		Clear(Context.SendSize);
		Clear(Context.RecvTimes);
		Clear(Context.RecvSize);

		iWillTcpEstablished := TRUE;
		iConnectRetryTimes := Context.ConnectRetryTimes;
		iConnectRetryInterval := MAX(UINT#100, Context.ConnectRetryInterval);
		iConnectTimeout := MAX(UINT#10, Context.ConnectTimeout);
		iWatchInterval := MAX(UINT#100, Context.WatchInterval);
		iOptionNodelay := Context.OptionNodelay;

		iState := STATE_WAIT;
		
	// STATE_WAIT
	5:
		IF Context.CtrlActive THEN
			iReturnState := iState + 1;
			iState := STATE_CONNECT;
		END_IF;
	6:
		IF iError THEN			
			Context.Error := TRUE;
			Context.ErrorID := iErrorID;
			Context.ErrorIDEx := iErrorIDEx;
			
			IF iConnectRetryTimes < 1 THEN
				iState := STATE_HALT;
			ELSE
				iReturnState := STATE_RECONNECT;
				iState := STATE_CLOSE;
			END_IF;
		ELSE
			iActive := TRUE;
			IF Context.UseSend THEN
				iStateSender := STATE_SENDER_INIT;
			END_IF;
			IF Context.UseWatcher THEN
				iStateWatcher := STATE_WATCHER_INIT;
			END_IF;
			
			iState := STATE_ACTIVE;
		END_IF;
			
	// STATE_HALT
	9:
		IF NOT (Context.CtrlActive AND Enable) THEN
			iState := STATE_FINALIZE;
		END_IF;
	
	// STATE_ACTIVE
	10:
		IF NOT (Context.CtrlActive AND Enable) THEN
			iState := STATE_FINALIZE;
		ELSIF iSenderError THEN
			Context.Error := TRUE;
			Context.ErrorID := iSenderErrorID;
			Context.ErrorIDEx := SHL(WORD_TO_DWORD(iSenderErrorID), 16) OR UINT_TO_DWORD(STATE_SENDER_SEND);
			iActive := FALSE;
			
			IF iConnectRetryTimes < 1 THEN
				iReturnState := STATE_HALT;
				iState := STATE_CLOSE;
			ELSE
				iReturnState := STATE_RECONNECT;
				iState := STATE_CLOSE;
			END_IF;
		ELSIF iWatcherError THEN
			Context.Error := TRUE;
			Context.ErrorID := iWatcherErrorID;
			Context.ErrorIDEx := SHL(WORD_TO_DWORD(iWatcherErrorID), 16) OR UINT_TO_DWORD(STATE_WATCHER_CHECK);
			iActive := FALSE;
			
			IF iConnectRetryTimes < 1 THEN
				iReturnState := STATE_HALT;
				iState := STATE_CLOSE;
			ELSE
				iReturnState := STATE_RECONNECT;
				iState := STATE_CLOSE;
			END_IF;
		ELSIF NOT iWillTcpEstablished THEN
			iActive := FALSE;
			
			IF iConnectRetryTimes < 1 THEN
				iReturnState := STATE_HALT;
				iState := STATE_CLOSE;
			ELSE
				iReturnState := STATE_RECONNECT;
				iState := STATE_CLOSE;
			END_IF;
		END_IF;		

	// STATE_RECONNECT
	20:
		iRetryTimes := iConnectRetryTimes;
		Timer(In:=FALSE,
			  PT:=iConnectRetryInterval,
			  TimerDat:=iRetryTimer,
			  Q=>iDoRetry);
		Context.Reconnecting := TRUE;
		
		Inc(iState);
	21:
		Timer(In:=TRUE,
			  PT:=iConnectRetryInterval,
			  TimerDat:=iRetryTimer,
			  Q=>iDoRetry);
		IF NOT (Context.CtrlActive AND Enable) THEN
			Context.Reconnecting := FALSE;
			
			iState := STATE_FINALIZE;
		ELSIF iDoRetry THEN
			iReturnState := iState + 1;
			iState := STATE_CONNECT;
		END_IF;
	22:
		IF iError THEN
			Dec(iRetryTimes);
			IF iRetryTimes < 1 THEN				
				iState := iState + 7;
			ELSE
				Timer(In:=FALSE,
					  PT:=iConnectRetryInterval,
					  TimerDat:=iRetryTimer,
					  Q=>iDoRetry);
				
				Dec(iState);
			END_IF;
		ELSE
			iState := iState + 7;
		END_IF;
	29:
		IF iError THEN
			Context.Error := TRUE;
			Context.ErrorID := iErrorID;
			Context.ErrorIDEx := iErrorIDEx;
			
			iState := STATE_HALT;
		ELSE
			Clear(Context.Error);
			Clear(Context.ErrorID);
			Clear(Context.ErrorIDEx);
			
			iActive := TRUE;
			IF Context.UseSend THEN
				iStateSender := STATE_SENDER_INIT;
			END_IF;
			IF Context.UseWatcher THEN
				iStateWatcher := STATE_WATCHER_INIT;
			END_IF;

			iState := STATE_ACTIVE;
		END_IF;
		Context.Reconnecting := FALSE;
		
	// STATE_CONNECT
	100:
		Clear(iError);
		Clear(iErrorID);
		Clear(iErrorIDEx);
		Timer(In:=FALSE,
			  PT:=iConnectTimeout,
			  TimerDat:=iTimeoutTimer);
		
		iSktTCPConnect.DstAdr := Context.Destination;
		iSktTCPConnect.DstTcpPort := Context.DestinationPort;
		iSktTCPConnect.SrcTcpPort := Context.Port;
		iSktTCPConnect.Execute := TRUE;

		Inc(iState);
	101:
		Timer(In:=TRUE,
			  PT:=iConnectTimeout,
			  TimerDat:=iTimeoutTimer,
			  Q=>iTimeout);
		IF iSktTCPConnect.Done OR iSktTCPConnect.Error THEN
			iSktTCPConnect.Execute := FALSE;
			
			IF iSktTCPConnect.Error THEN
				iError := TRUE;
				iErrorID := iSktTCPConnect.ErrorID;
				iErrorIDEx := SHL(WORD_TO_DWORD(iErrorID), 16) OR UINT_TO_DWORD(iState);
				
				iState := iState + 8;
			ELSE
				iSocket := iSktTCPConnect.Socket;
				Context.Socket := iSocket;

				Inc(iState);
			END_IF;
		ELSIF iTimeout THEN
			iSktTCPConnect.Execute := FALSE;
			
			iError := TRUE;
			iErrorID := WORD#16#2006; // Socket timeout.
			iErrorIDEx := SHL(WORD_TO_DWORD(iErrorID), 16) OR UINT_TO_DWORD(iState);
			
			iState := iState + 8;
		END_IF;
	102:
		IF NOT Context.UseTcpSocketOption THEN
			iState := iState + 3;
		ELSE
			Inc(iState);
		END_IF;
	103:
		iSktSetOption(Execute:=FALSE,
					  OptionType:=_eSKT_OPTION_TYPE#_TCP_NODELAY,
					  OptionParam:=iOptionNodelay);

		Inc(iState);
	104:
		iSktSetOption(Execute:=TRUE,
					  Socket:=iSocket,
					  OptionType:=_eSKT_OPTION_TYPE#_TCP_NODELAY,
					  OptionParam:=iOptionNodelay);

		IF iSktSetOption.Done OR iSktSetOption.Error THEN
			iSktSetOption.Execute := FALSE;

			IF iSktSetOption.Error THEN
				iError := TRUE;
				iErrorID := iSktSetOption.ErrorID;
				iErrorIDEx := SHL(WORD_TO_DWORD(iErrorID), 16) OR UINT_TO_DWORD(iState);
				
				iState := iState + 5;
			ELSE
				Inc(iState);
			END_IF;
		END_IF;
	105:
		iSktTLSConnect.Socket := iSocket;
		iSktTLSConnect.TLSSessionName := Context.TLSSessionName;
		iSktTLSConnect.Execute := TRUE;
		
		Inc(iState);
	106:
		IF iSktTLSConnect.Done OR iSktTLSConnect.Error THEN
			iSktTLSConnect.Execute := FALSE;
			
			IF iSktTLSConnect.Error THEN
				iError := TRUE;
				iErrorID := iSktTLSConnect.ErrorID;
				iErrorIDEx := SHL(WORD_TO_DWORD(iErrorID), 16) OR UINT_TO_DWORD(iState);	
			ELSE
				iTLSHandle := iSktTLSConnect.Handle;
				Context.TLSHandle := iTLSHandle;
			END_IF;
			
			iState := iState + 3;
		END_IF;
	109:
		Context.Connected := NOT iError;
		
		iState := iReturnState;

	// STATE_CLOSE
	110:
		Clear(iError);
		Clear(iErrorID);
		Clear(iErrorIDEx);
	
		iSktTLSDisconnect.Handle := iTLSHandle;
		iSktTLSDisconnect.Execute := TRUE;
		
		Inc(iState);
	111:
		IF iSktTLSDisconnect.Done OR iSktTLSDisconnect.Error THEN
			iSktTLSDisconnect.Execute := FALSE;
			
			IF iSktTLSDisconnect.Error THEN
				iError := TRUE;
				iErrorID := iSktTLSDisconnect.ErrorID;
				iErrorIDEx := SHL(WORD_TO_DWORD(iErrorID), 16) OR UINT_TO_DWORD(iState);
			END_IF;
			
			Inc(iState);
		END_IF;
	112:
		iSktClose.Socket := iSocket;
		iSktClose.Execute := TRUE;
		
		Inc(iState);
	113:
		IF iSktClose.Done OR iSktClose.Error THEN
			iSktClose.Execute := FALSE;
			
			IF iSktClose.Error AND NOT iError THEN
				iError := TRUE;
				iErrorID := iSktClose.ErrorID;
				iErrorIDEx := SHL(WORD_TO_DWORD(iErrorID), 16) OR UINT_TO_DWORD(iState);
			END_IF;
			
			iState := iState + 6;
		END_IF;
	119:
		Context.Connected := FALSE;
		
		iState := iReturnState;
		
	// STATE_FINALIZE
	900:
		iActive := FALSE;
		
		Inc(iState);
	901:
		IF iStateSender = STATE_SENDER_DONE THEN
			IF iSenderError AND NOT Context.Error THEN
				Context.Error := TRUE;
				Context.ErrorID := iSenderErrorID;
				Context.ErrorIDEx := SHL(WORD_TO_DWORD(iSenderErrorID), 16) OR UINT_TO_DWORD(iState);
			END_IF;
			
			iState := iState + 2;
		END_IF;
	903:
		IF iStateWatcher = STATE_WATCHER_DONE THEN
			IF iWatcherError AND NOT Context.Error THEN
				Context.Error := TRUE;
				Context.ErrorID := iWatcherErrorID;
				Context.ErrorIDEx := SHL(WORD_TO_DWORD(iWatcherErrorID), 16) OR UINT_TO_DWORD(iState);
			END_IF;
			
			Inc(iState);
		END_IF;
	904:
		IF Context.Connected THEN
			iReturnState := iState + 1;
			iState := STATE_CLOSE;
		ELSE
			iState := iState + 5;
		END_IF;
	905:
		IF iError AND NOT Context.Error THEN
			Context.Error := TRUE;
			Context.ErrorID := iErrorID;
			Context.ErrorIDEx := iErrorIDEx;
		END_IF;
		
		iState := iState + 4;
	909:
		iState := STATE_DONE;
	
	// STATE_DONE
	1000:
		Done := TRUE;
		Busy := FALSE;
		
		Inc(iState);
END_CASE;

CASE iStateSender OF
	// STATE_SENDER_INIT
	0:
		iSktTLSWrite.Execute := FALSE;

		Clear(iSenderError);
		Clear(iSenderErrorID);
		
		iStateSender := STATE_SENDER_ACTIVE;
				
	// STATE_SENDER_ACTIVE
	10:
		IF NOT iActive THEN
			iStateSender := STATE_SENDER_DONE;
		ELSIF \\stfreakjp\buf\RingBuffer_isReadable(
								  Context:=SendBufferContext)
		THEN
			iStateSender := STATE_SENDER_SEND;
		END_IF;
	
	// STATE_SENDER_SEND
	200:
		IF Context.CtrlAllowSend THEN
			\\stfreakjp\buf\RingBuffer_peekFully(
								Context:=SendBufferContext,
								Buffer:=SendBuffer,
								Out:=iSendData,
								Head:=0,
								ReadSize=>iSendDataSize);
			
			IF iSendDataSize < 1 THEN
				iStateSender := STATE_SENDER_ACTIVE;
			ELSE
				iSktTLSWrite.Handle := iTLSHandle;
				iSktTLSWrite.SendDatSize := iSendDataSize;
				iSktTLSWrite.Execute := TRUE;
				
				Inc(iStateSender);
			END_IF;
		ELSIF NOT iActive THEN
			iStateSender := STATE_SENDER_DONE;
		END_IF;
	201:
		IF iSktTLSWrite.Done OR iSktTLSWrite.Error THEN
			iSktTLSWrite.Execute := FALSE;
			
			IF iSktTLSWrite.Error THEN
				iSenderErrorID := iSktTLSWrite.ErrorID;
				CASE WORD_TO_UINT(iSenderErrorID) OF
					// Socket communication resource over.
					16#2008:
						iSenderWaitTick
							:= MAX(UINT#10, TO_UINT(iSendDataSize MOD 50));
						
						Inc(iStateSender);
				ELSE
					iSenderError := TRUE;
					
					iStateSender := STATE_SENDER_DONE;
				END_CASE;
			ELSE
				\\stfreakjp\buf\RingBuffer_consume(
									Context:=SendBufferContext,
									Buffer:=SendBuffer,
									Size:=iSendDataSize);
				
				Context.SendSize := Context.SendSize + iSendDataSize;
				Inc(Context.SendTimes);
				
				Dec(iStateSender);
			END_IF;
		END_IF;
	202:
		Dec(iSenderWaitTick);
		IF NOT iActive THEN
			iSenderError := TRUE;

			iStateSender := STATE_SENDER_DONE;
		ELSIF NOT Context.CtrlAllowSend THEN
			iStateSender := iStateSender - 2;
		ELSIF iSenderWaitTick < 1 THEN
			iSktTLSWrite.Execute := TRUE;
			
			Dec(iStateSender);
		END_IF;
	
	// STATE_SENDER_DONE
	// 1000:
END_CASE;

CASE iStateWatcher OF
	// STATE_WATCHER_INIT
	0:
		iSktGetTCPStatus.Execute := FALSE;
		
		Clear(iWatcherError);
		Clear(iWatcherErrorID);

		Timer(In:=FALSE,
			  PT:=iWatchInterval,
			  TimerDat:=iWatchTimer);
		
		iStateWatcher := STATE_WATCHER_ACTIVE;
		
	// STATE_WATCHER_ACTIVE
	10:
		Timer(In:=TRUE,
			  PT:=iWatchInterval,
			  TimerDat:=iWatchTimer,
			  Q=>iWatchDoCheck);
		IF NOT iActive THEN
			iStateWatcher := STATE_WATCHER_DONE;
		ELSIF iWatchDoCheck THEN
			iStateWatcher := STATE_WATCHER_CHECK;
		END_IF;
	
	// STATE_WATCHER_CHECK
	400:
		iSktGetTCPStatus.Socket := iSocket;
		iSktGetTCPStatus.Execute := TRUE;
		
		Inc(iStateWatcher);
	401:
		IF iSktGetTCPStatus.Done OR iSktGetTCPStatus.Error THEN
			iSktGetTCPStatus.Execute := FALSE;
			
			IF iSktGetTCPStatus.Error THEN
				iWatcherError := TRUE;
				iWatcherErrorID := iSktGetTCPStatus.ErrorID;
				
				iStateWatcher := STATE_WATCHER_DONE;
			ELSE
				iTcpStatus := iSktGetTCPStatus.TcpStatus;
				CASE iTcpStatus OF
					_eCONNECTION_STATE#_ESTABLISHED:
						iWillTcpEstablished := TRUE;
				ELSE
					iWillTcpEstablished := FALSE;
				END_CASE;
				
				Timer(In:=FALSE,
					  PT:=iWatchInterval,
					  TimerDat:=iWatchTimer);
				
				iStateWatcher := STATE_WATCHER_ACTIVE;
			END_IF;
		END_IF;
	
	// STATE_WATCHER_DONE
	// 1000:
END_CASE;

iSktTCPConnect();
iSktClose();
iSktGetTCPStatus();
iSktTLSConnect();
iSktTLSDisconnect();
iSktTLSWrite(SendDat:=iSendData[0]);

Context.Active := iActive;
Context.Busy := Busy;
END_FUNCTION_BLOCK

FUNCTION_BLOCK stfreakjp\net\TlsRecvClient
(* TLS client that performs sending and receiving operations. *)
VAR
    iSktTCPConnect : SktTCPConnect;
    iSktClose : SktClose;
    iSktGetTCPStatus : SktGetTCPStatus;
    iSktSetOption : SktSetOption;
    iSktTLSConnect : SktTLSConnect;
    iSktTLSDisconnect : SktTLSDisconnect;
    iSktTLSRead : SktTLSRead;
END_VAR
VAR CONSTANT
    STATE_INIT : UINT := 0;
    STATE_WAIT : UINT := 5;
    STATE_HALT : UINT := 9;
    STATE_ACTIVE : UINT := 10;
    STATE_RECONNECT : UINT := 20;
    STATE_CONNECT : UINT := 100;
    STATE_CLOSE : UINT := 110;
    STATE_CHANGE_DESTINATION : UINT := 120;
    STATE_FINALIZE : UINT := 900;
    STATE_DONE : UINT := 1000;
    STATE_RECEIVER_INIT : UINT := 0;
    STATE_RECEIVER_WAIT : UINT := 5;
    STATE_RECEIVER_ACTIVE : UINT := 10;
    STATE_RECEIVER_RECV : UINT := 300;
    STATE_RECEIVER_DONE : UINT := 1000;
    STATE_WATCHER_INIT : UINT := 0;
    STATE_WATCHER_ACTIVE : UINT := 10;
    STATE_WATCHER_CHECK : UINT := 400;
    STATE_WATCHER_DONE : UINT := 1000;
END_VAR
VAR
    iState : UINT := 1001;
    iReturnState : UINT;
    iSocket : _sSOCKET;
    iTLSHandle : DWORD;
    iActive : BOOL;
    iError : BOOL;
    iErrorID : WORD;
    iErrorIDEx : DWORD;
    iConnectRetryTimes : UINT;
    iConnectRetryInterval : UINT;
    iConnectTimeout : UINT;
    iTimeoutTimer : _sTimer;
    iTimeout : BOOL;
    iWatchInterval : UINT;
    iWillTcpEstablished : BOOL;
    iTcpStatus : _eCONNECTION_STATE;
    iOptionNodelay : BOOL;
    iRetryTimes : UINT;
    iRetryInterval : UINT;
    iRetryTimer : _sTimer;
    iDoRetry : BOOL;
    iStateReceiver : UINT := 1000;
    iRecvData : ARRAY[0..1999] OF BYTE;
    iRecvDataSize : UINT;
    iReceiverError : BOOL;
    iReceiverErrorID : WORD;
    iReceiverWaitTick : UINT;
    iStateWatcher : UINT := 1000;
    iWatcherError : BOOL;
    iWatcherErrorID : WORD;
    iWatchTimer : _sTimer;
    iWatchDoCheck : BOOL;
END_VAR
VAR_INPUT
    Enable : BOOL;  (* Enable TlsClient FB. *)
END_VAR
VAR_IN_OUT
    Context : stfreakjp\net\TlsClientContext;  (* TlsClientContext to process. *)
    RecvBufferContext : stfreakjp\buf\RingBufferContext;  (* RingBufferContext for the received data. *)
    RecvBuffer : ARRAY[*] OF BYTE;  (* Buffer for received data. *)
END_VAR
VAR_OUTPUT
    Busy : BOOL;  (* Whether the TlsClient is running. *)
    Done : BOOL;  (* Whether the TlsClient has completed processing. *)
END_VAR
(*

TLS client that performs receiving operations.


受信処理を行うTLSクライアント。

(c) 2025 KITA Munemitsu

*)

Done := FALSE;
IF Enable AND NOT Busy THEN
	iState := STATE_INIT;
	
	Busy := TRUE;
END_IF;

CASE iState OF
	// STATE_INIT
	0:
		iSktTCPConnect.Execute := FALSE;
		iSktClose.Execute := FALSE;
		iSktGetTCPStatus.Execute := FALSE;
		iSktTLSConnect.Execute := FALSE;
		iSktTLSDisconnect.Execute := FALSE;
		iSktTLSRead.Execute := FALSE;

		Clear(iActive);
		Clear(iSocket);
		Clear(iTLSHandle);
		Clear(iError);
		Clear(iErrorID);
		Clear(iErrorIDEx);
		
		Clear(Context.Active);
		Clear(Context.Busy);
		Clear(Context.Error);
		Clear(Context.ErrorID);
		Clear(Context.ErrorIDEx);
		Clear(Context.Connected);
		Clear(Context.Reconnecting);
		Clear(Context.Socket);
		Clear(Context.TLSHandle);
		Clear(Context.SendTimes);
		Clear(Context.SendSize);
		Clear(Context.RecvTimes);
		Clear(Context.RecvSize);

		iWillTcpEstablished := TRUE;
		iConnectRetryTimes := Context.ConnectRetryTimes;
		iConnectRetryInterval := MAX(UINT#100, Context.ConnectRetryInterval);
		iConnectTimeout := MAX(UINT#10, Context.ConnectTimeout);
		iWatchInterval := MAX(UINT#100, Context.WatchInterval);
		iOptionNodelay := Context.OptionNodelay;

		iState := STATE_WAIT;
		
	// STATE_WAIT
	5:
		IF Context.CtrlActive THEN
			iReturnState := iState + 1;
			iState := STATE_CONNECT;
		END_IF;
	6:
		IF iError THEN			
			Context.Error := TRUE;
			Context.ErrorID := iErrorID;
			Context.ErrorIDEx := iErrorIDEx;
			
			IF iConnectRetryTimes < 1 THEN
				iState := STATE_HALT;
			ELSE
				iReturnState := STATE_RECONNECT;
				iState := STATE_CLOSE;
			END_IF;
		ELSE
			iActive := TRUE;
			IF Context.UseRecv THEN
				iStateReceiver := STATE_RECEIVER_INIT;
			END_IF;
			IF Context.UseWatcher THEN
				iStateWatcher := STATE_WATCHER_INIT;
			END_IF;
			
			iState := STATE_ACTIVE;
		END_IF;
			
	// STATE_HALT
	9:
		IF NOT (Context.CtrlActive AND Enable) THEN
			iState := STATE_FINALIZE;
		END_IF;
	
	// STATE_ACTIVE
	10:
		IF NOT (Context.CtrlActive AND Enable) THEN
			iState := STATE_FINALIZE;
		ELSIF iReceiverError THEN
			Context.Error := TRUE;
			Context.ErrorID := iReceiverErrorID;
			Context.ErrorIDEx := SHL(WORD_TO_DWORD(iReceiverErrorID), 16) OR UINT_TO_DWORD(STATE_RECEIVER_RECV);
			iActive := FALSE;
			
			IF iConnectRetryTimes < 1 THEN
				iReturnState := STATE_HALT;
				iState := STATE_CLOSE;
			ELSE
				iReturnState := STATE_RECONNECT;
				iState := STATE_CLOSE;
			END_IF;
		ELSIF iWatcherError THEN
			Context.Error := TRUE;
			Context.ErrorID := iWatcherErrorID;
			Context.ErrorIDEx := SHL(WORD_TO_DWORD(iWatcherErrorID), 16) OR UINT_TO_DWORD(STATE_WATCHER_CHECK);
			iActive := FALSE;
			
			IF iConnectRetryTimes < 1 THEN
				iReturnState := STATE_HALT;
				iState := STATE_CLOSE;
			ELSE
				iReturnState := STATE_RECONNECT;
				iState := STATE_CLOSE;
			END_IF;
		ELSIF NOT iWillTcpEstablished THEN
			iActive := FALSE;
			
			IF iConnectRetryTimes < 1 THEN
				iReturnState := STATE_HALT;
				iState := STATE_CLOSE;
			ELSE
				iReturnState := STATE_RECONNECT;
				iState := STATE_CLOSE;
			END_IF;
		END_IF;		

	// STATE_RECONNECT
	20:
		iRetryTimes := iConnectRetryTimes;
		Timer(In:=FALSE,
			  PT:=iConnectRetryInterval,
			  TimerDat:=iRetryTimer,
			  Q=>iDoRetry);
		Context.Reconnecting := TRUE;
		
		Inc(iState);
	21:
		Timer(In:=TRUE,
			  PT:=iConnectRetryInterval,
			  TimerDat:=iRetryTimer,
			  Q=>iDoRetry);
		IF NOT (Context.CtrlActive AND Enable) THEN
			Context.Reconnecting := FALSE;
			
			iState := STATE_FINALIZE;
		ELSIF iDoRetry THEN
			iReturnState := iState + 1;
			iState := STATE_CONNECT;
		END_IF;
	22:
		IF iError THEN
			Dec(iRetryTimes);
			IF iRetryTimes < 1 THEN				
				iState := iState + 7;
			ELSE
				Timer(In:=FALSE,
					  PT:=iConnectRetryInterval,
					  TimerDat:=iRetryTimer,
					  Q=>iDoRetry);
				
				Dec(iState);
			END_IF;
		ELSE
			iState := iState + 7;
		END_IF;
	29:
		IF iError THEN
			Context.Error := TRUE;
			Context.ErrorID := iErrorID;
			Context.ErrorIDEx := iErrorIDEx;
			
			iState := STATE_HALT;
		ELSE
			Clear(Context.Error);
			Clear(Context.ErrorID);
			Clear(Context.ErrorIDEx);
			
			iActive := TRUE;
			IF Context.UseRecv THEN
				iStateReceiver := STATE_RECEIVER_INIT;
			END_IF;
			IF Context.UseWatcher THEN
				iStateWatcher := STATE_WATCHER_INIT;
			END_IF;

			iState := STATE_ACTIVE;
		END_IF;
		Context.Reconnecting := FALSE;
		
	// STATE_CONNECT
	100:
		Clear(iError);
		Clear(iErrorID);
		Clear(iErrorIDEx);
		Timer(In:=FALSE,
			  PT:=iConnectTimeout,
			  TimerDat:=iTimeoutTimer);
		
		iSktTCPConnect.DstAdr := Context.Destination;
		iSktTCPConnect.DstTcpPort := Context.DestinationPort;
		iSktTCPConnect.SrcTcpPort := Context.Port;
		iSktTCPConnect.Execute := TRUE;

		Inc(iState);
	101:
		Timer(In:=TRUE,
			  PT:=iConnectTimeout,
			  TimerDat:=iTimeoutTimer,
			  Q=>iTimeout);
		IF iSktTCPConnect.Done OR iSktTCPConnect.Error THEN
			iSktTCPConnect.Execute := FALSE;
			
			IF iSktTCPConnect.Error THEN
				iError := TRUE;
				iErrorID := iSktTCPConnect.ErrorID;
				iErrorIDEx := SHL(WORD_TO_DWORD(iErrorID), 16) OR UINT_TO_DWORD(iState);
				
				iState := iState + 8;
			ELSE
				iSocket := iSktTCPConnect.Socket;
				Context.Socket := iSocket;

				Inc(iState);
			END_IF;
		ELSIF iTimeout THEN
			iSktTCPConnect.Execute := FALSE;
			
			iError := TRUE;
			iErrorID := WORD#16#2006; // Socket timeout.
			iErrorIDEx := SHL(WORD_TO_DWORD(iErrorID), 16) OR UINT_TO_DWORD(iState);
			
			iState := iState + 8;
		END_IF;
	102:
		IF NOT Context.UseTcpSocketOption THEN
			iState := iState + 3;
		ELSE
			Inc(iState);
		END_IF;
	103:
		iSktSetOption(Execute:=FALSE,
					  OptionType:=_eSKT_OPTION_TYPE#_TCP_NODELAY,
					  OptionParam:=iOptionNodelay);

		Inc(iState);
	104:
		iSktSetOption(Execute:=TRUE,
					  Socket:=iSocket,
					  OptionType:=_eSKT_OPTION_TYPE#_TCP_NODELAY,
					  OptionParam:=iOptionNodelay);

		IF iSktSetOption.Done OR iSktSetOption.Error THEN
			iSktSetOption.Execute := FALSE;

			IF iSktSetOption.Error THEN
				iError := TRUE;
				iErrorID := iSktSetOption.ErrorID;
				iErrorIDEx := SHL(WORD_TO_DWORD(iErrorID), 16) OR UINT_TO_DWORD(iState);
				
				iState := iState + 5;
			ELSE
				Inc(iState);
			END_IF;
		END_IF;
	105:
		iSktTLSConnect.Socket := iSocket;
		iSktTLSConnect.TLSSessionName := Context.TLSSessionName;
		iSktTLSConnect.Execute := TRUE;
		
		Inc(iState);
	106:
		IF iSktTLSConnect.Done OR iSktTLSConnect.Error THEN
			iSktTLSConnect.Execute := FALSE;
			
			IF iSktTLSConnect.Error THEN
				iError := TRUE;
				iErrorID := iSktTLSConnect.ErrorID;
				iErrorIDEx := SHL(WORD_TO_DWORD(iErrorID), 16) OR UINT_TO_DWORD(iState);	
			ELSE
				iTLSHandle := iSktTLSConnect.Handle;
				Context.TLSHandle := iTLSHandle;
			END_IF;
			
			iState := iState + 3;
		END_IF;
	109:
		Context.Connected := NOT iError;
		
		iState := iReturnState;

	// STATE_CLOSE
	110:
		Clear(iError);
		Clear(iErrorID);
		Clear(iErrorIDEx);
	
		iSktTLSDisconnect.Handle := iTLSHandle;
		iSktTLSDisconnect.Execute := TRUE;
		
		Inc(iState);
	111:
		IF iSktTLSDisconnect.Done OR iSktTLSDisconnect.Error THEN
			iSktTLSDisconnect.Execute := FALSE;
			
			IF iSktTLSDisconnect.Error THEN
				iError := TRUE;
				iErrorID := iSktTLSDisconnect.ErrorID;
				iErrorIDEx := SHL(WORD_TO_DWORD(iErrorID), 16) OR UINT_TO_DWORD(iState);
			END_IF;
			
			Inc(iState);
		END_IF;
	112:
		iSktClose.Socket := iSocket;
		iSktClose.Execute := TRUE;
		
		Inc(iState);
	113:
		IF iSktClose.Done OR iSktClose.Error THEN
			iSktClose.Execute := FALSE;
			
			IF iSktClose.Error AND NOT iError THEN
				iError := TRUE;
				iErrorID := iSktClose.ErrorID;
				iErrorIDEx := SHL(WORD_TO_DWORD(iErrorID), 16) OR UINT_TO_DWORD(iState);
			END_IF;
			
			iState := iState + 6;
		END_IF;
	119:
		Context.Connected := FALSE;
		
		iState := iReturnState;
		
	// STATE_FINALIZE
	900:
		iActive := FALSE;
		
		iState := iState + 2;
	902:
		IF iStateReceiver = STATE_RECEIVER_DONE THEN
			IF iReceiverError AND NOT Context.Error THEN
				Context.Error := TRUE;
				Context.ErrorID := iReceiverErrorID;
				Context.ErrorIDEx := SHL(WORD_TO_DWORD(iReceiverErrorID), 16) OR UINT_TO_DWORD(iState);
			END_IF;
			
			Inc(iState);
		END_IF;
	903:
		IF iStateWatcher = STATE_WATCHER_DONE THEN
			IF iWatcherError AND NOT Context.Error THEN
				Context.Error := TRUE;
				Context.ErrorID := iWatcherErrorID;
				Context.ErrorIDEx := SHL(WORD_TO_DWORD(iWatcherErrorID), 16) OR UINT_TO_DWORD(iState);
			END_IF;
			
			Inc(iState);
		END_IF;
	904:
		IF Context.Connected THEN
			iReturnState := iState + 1;
			iState := STATE_CLOSE;
		ELSE
			iState := iState + 5;
		END_IF;
	905:
		IF iError AND NOT Context.Error THEN
			Context.Error := TRUE;
			Context.ErrorID := iErrorID;
			Context.ErrorIDEx := iErrorIDEx;
		END_IF;
		
		iState := iState + 4;
	909:
		iState := STATE_DONE;
	
	// STATE_DONE
	1000:
		Done := TRUE;
		Busy := FALSE;
		
		Inc(iState);
END_CASE;

CASE iStateReceiver OF
	// STATE_RECEIVER_INIT
	0:
		iSktTLSRead.Execute := FALSE;

		Clear(iReceiverError);
		Clear(iReceiverErrorID);
		
		iStateReceiver := STATE_RECEIVER_ACTIVE;
				
	// STATE_RECEIVER_ACTIVE
	10:
		IF NOT iActive THEN
			iStateReceiver := STATE_RECEIVER_DONE;
		ELSIF \\stfreakjp\buf\RingBuffer_isWritable(
								  Context:=RecvBufferContext)
		THEN
			iStateReceiver := STATE_RECEIVER_RECV;
		END_IF;
	
	// STATE_RECEIVER_RECV
	300:
		IF Context.CtrlAllowRecv THEN
			iSktTLSRead.TimeOut := 0;
			iSktTLSRead.Handle := iTLSHandle;
			iSktTLSRead.Execute := TRUE;
		
			Inc(iStateReceiver);
		ELSIF NOT iActive THEN
			iStateReceiver := STATE_RECEIVER_DONE;
		END_IF;
	301:
		IF NOT iActive THEN
			iSktTLSRead.Execute := FALSE;
			
			iStateReceiver := STATE_RECEIVER_DONE;
		ELSIF NOT Context.CtrlAllowRecv THEN
			iSktTLSRead.Execute := FALSE;
			
			Dec(iStateReceiver);
		ELSIF iSktTLSRead.Done OR iSktTLSRead.Error THEN
			iSktTLSRead.Execute := FALSE;
			
			IF iSktTLSRead.Error THEN
				iReceiverErrorID := iSktTLSRead.ErrorID;
				CASE WORD_TO_UINT(iReceiverErrorID) OF
					// Socket communication resource over.
					16#2008:
						iReceiverWaitTick := UINT#10;
						
						iStateReceiver := iStateReceiver + 2;
				ELSE
					iReceiverError := TRUE;
					
					iStateReceiver := STATE_RECEIVER_DONE;
				END_CASE;
			ELSE
				iRecvDataSize := iSktTLSRead.RcvSize;
				Context.RecvSize := Context.RecvSize + iRecvDataSize;
				Inc(Context.RecvTimes);
				
				IF \\stfreakjp\buf\RingBuffer_write(
									   Context:=RecvBufferContext,
									   Buffer:=RecvBuffer,
									   In:=iRecvData,
									   Head:=0,
									   Size:=iRecvDataSize)
				THEN					
					Dec(iStateReceiver);
				ELSE					
					Inc(iStateReceiver);
				END_IF;
			END_IF;
		END_IF;
	302:
		IF NOT iActive THEN
			iStateReceiver := STATE_RECEIVER_DONE;
		ELSIF \\stfreakjp\buf\RingBuffer_write(
								  Context:=RecvBufferContext,
								  Buffer:=RecvBuffer,
								  In:=iRecvData,
								  Head:=0,
								  Size:=iRecvDataSize)
		THEN
			iStateReceiver := iStateReceiver - 2;
		END_IF;
	303:
		Dec(iReceiverWaitTick);
		IF NOT iActive THEN
			iReceiverError := TRUE;

			iStateReceiver := STATE_RECEIVER_DONE;
		ELSIF iReceiverWaitTick < 1 THEN
			iStateReceiver := iStateReceiver - 3;
		END_IF;
	
	// STATE_RECEIVER_DONE
	// 1000:
END_CASE;

CASE iStateWatcher OF
	// STATE_WATCHER_INIT
	0:
		iSktGetTCPStatus.Execute := FALSE;
		
		Clear(iWatcherError);
		Clear(iWatcherErrorID);

		Timer(In:=FALSE,
			  PT:=iWatchInterval,
			  TimerDat:=iWatchTimer);
		
		iStateWatcher := STATE_WATCHER_ACTIVE;
		
	// STATE_WATCHER_ACTIVE
	10:
		Timer(In:=TRUE,
			  PT:=iWatchInterval,
			  TimerDat:=iWatchTimer,
			  Q=>iWatchDoCheck);
		IF NOT iActive THEN
			iStateWatcher := STATE_WATCHER_DONE;
		ELSIF iWatchDoCheck THEN
			iStateWatcher := STATE_WATCHER_CHECK;
		END_IF;
	
	// STATE_WATCHER_CHECK
	400:
		iSktGetTCPStatus.Socket := iSocket;
		iSktGetTCPStatus.Execute := TRUE;
		
		Inc(iStateWatcher);
	401:
		IF iSktGetTCPStatus.Done OR iSktGetTCPStatus.Error THEN
			iSktGetTCPStatus.Execute := FALSE;
			
			IF iSktGetTCPStatus.Error THEN
				iWatcherError := TRUE;
				iWatcherErrorID := iSktGetTCPStatus.ErrorID;
				
				iStateWatcher := STATE_WATCHER_DONE;
			ELSE
				iTcpStatus := iSktGetTCPStatus.TcpStatus;
				CASE iTcpStatus OF
					_eCONNECTION_STATE#_ESTABLISHED:
						iWillTcpEstablished := TRUE;
				ELSE
					iWillTcpEstablished := FALSE;
				END_CASE;
				
				Timer(In:=FALSE,
					  PT:=iWatchInterval,
					  TimerDat:=iWatchTimer);
				
				iStateWatcher := STATE_WATCHER_ACTIVE;
			END_IF;
		END_IF;
	
	// STATE_WATCHER_DONE
	// 1000:
END_CASE;

iSktTCPConnect();
iSktClose();
iSktGetTCPStatus();
iSktTLSConnect();
iSktTLSDisconnect();
iSktTLSRead(RcvDat:=iRecvData[0]);

Context.Active := iActive;
Context.Busy := Busy;
END_FUNCTION_BLOCK